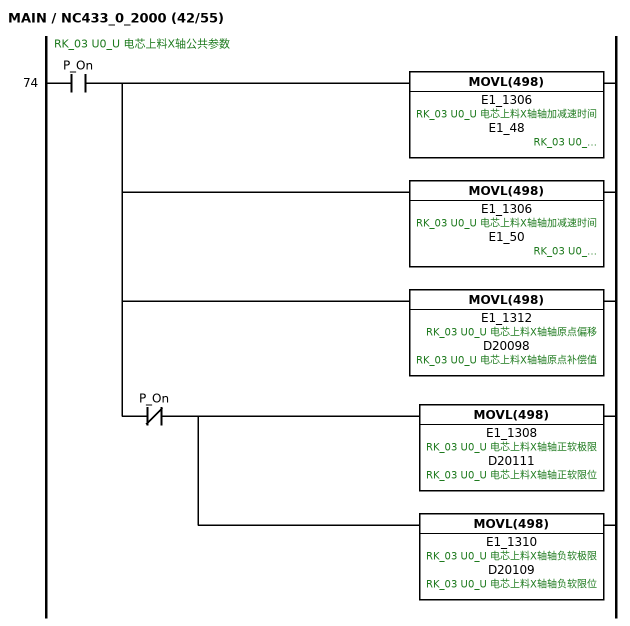
; [picture p96: MAIN / NC433_0_2000, rungs 74-74]
; rung 74: RK_03 U0_U 电芯上料X轴公共参数
LD P_On
MOVL(498) E1_1306 E1_48  ; RK_03 U0_U 电芯上料X轴轴加减速时间, RK_03 U0_U 电芯上料X轴轴直接操作加速时间
MOVL(498) E1_1306 E1_50  ; RK_03 U0_U 电芯上料X轴轴加减速时间, RK_03 U0_U 电芯上料X轴轴直接操作减速时间
MOVL(498) E1_1312 D20098  ; RK_03 U0_U 电芯上料X轴轴原点偏移, RK_03 U0_U 电芯上料X轴轴原点补偿值
ANDNOT P_On
MOVL(498) E1_1308 D20111  ; RK_03 U0_U 电芯上料X轴轴正软极限, RK_03 U0_U 电芯上料X轴轴正软限位
MOVL(498) E1_1310 D20109  ; RK_03 U0_U 电芯上料X轴轴负软极限, RK_03 U0_U 电芯上料X轴轴负软限位

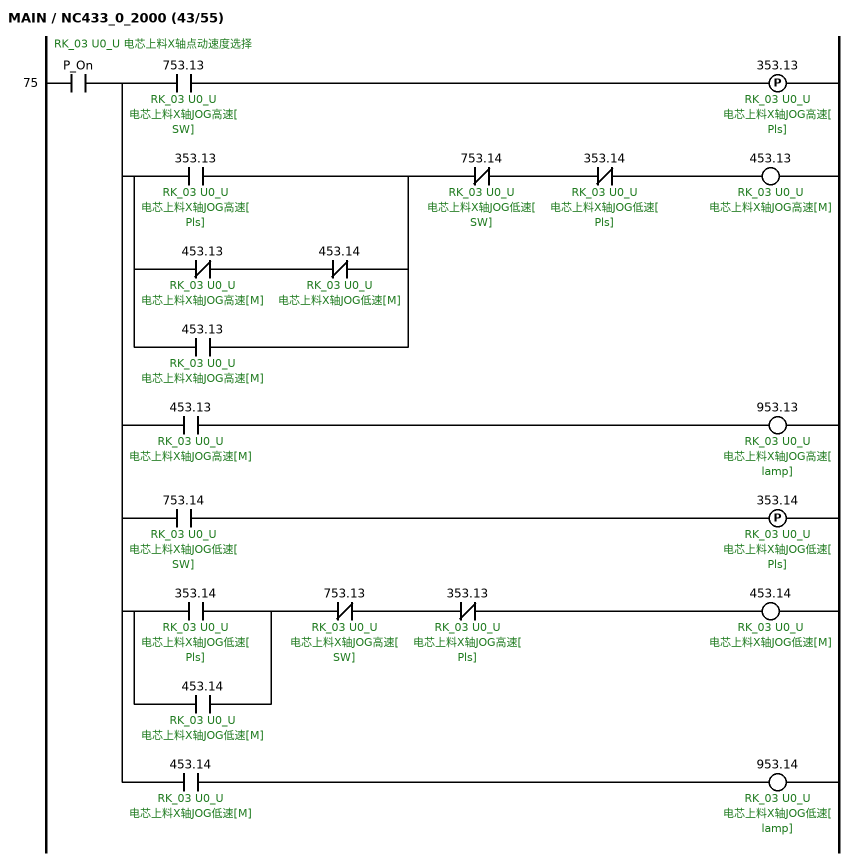
; rung 75: RK_03 U0_U 电芯上料X轴点动速度选择
LD P_On
OUT TR0
AND 753.13  ; RK_03 U0_U 电芯上料X轴JOG高速[SW]
DIFU(013) 353.13  ; RK_03 U0_U 电芯上料X轴JOG高速[Pls]
LD TR0
LD 353.13  ; RK_03 U0_U 电芯上料X轴JOG高速[Pls]
LDNOT 453.13  ; RK_03 U0_U 电芯上料X轴JOG高速[M]
ANDNOT 453.14  ; RK_03 U0_U 电芯上料X轴JOG低速[M]
ORLD
OR 453.13  ; RK_03 U0_U 电芯上料X轴JOG高速[M]
ANDLD
ANDNOT 753.14  ; RK_03 U0_U 电芯上料X轴JOG低速[SW]
ANDNOT 353.14  ; RK_03 U0_U 电芯上料X轴JOG低速[Pls]
OUT 453.13  ; RK_03 U0_U 电芯上料X轴JOG高速[M]
LD TR0
AND 453.13  ; RK_03 U0_U 电芯上料X轴JOG高速[M]
OUT 953.13  ; RK_03 U0_U 电芯上料X轴JOG高速[lamp]
LD TR0
AND 753.14  ; RK_03 U0_U 电芯上料X轴JOG低速[SW]
DIFU(013) 353.14  ; RK_03 U0_U 电芯上料X轴JOG低速[Pls]
LD TR0
LD 353.14  ; RK_03 U0_U 电芯上料X轴JOG低速[Pls]
OR 453.14  ; RK_03 U0_U 电芯上料X轴JOG低速[M]
ANDLD
ANDNOT 753.13  ; RK_03 U0_U 电芯上料X轴JOG高速[SW]
ANDNOT 353.13  ; RK_03 U0_U 电芯上料X轴JOG高速[Pls]
OUT 453.14  ; RK_03 U0_U 电芯上料X轴JOG低速[M]
LD TR0
AND 453.14  ; RK_03 U0_U 电芯上料X轴JOG低速[M]
OUT 953.14  ; RK_03 U0_U 电芯上料X轴JOG低速[lamp]

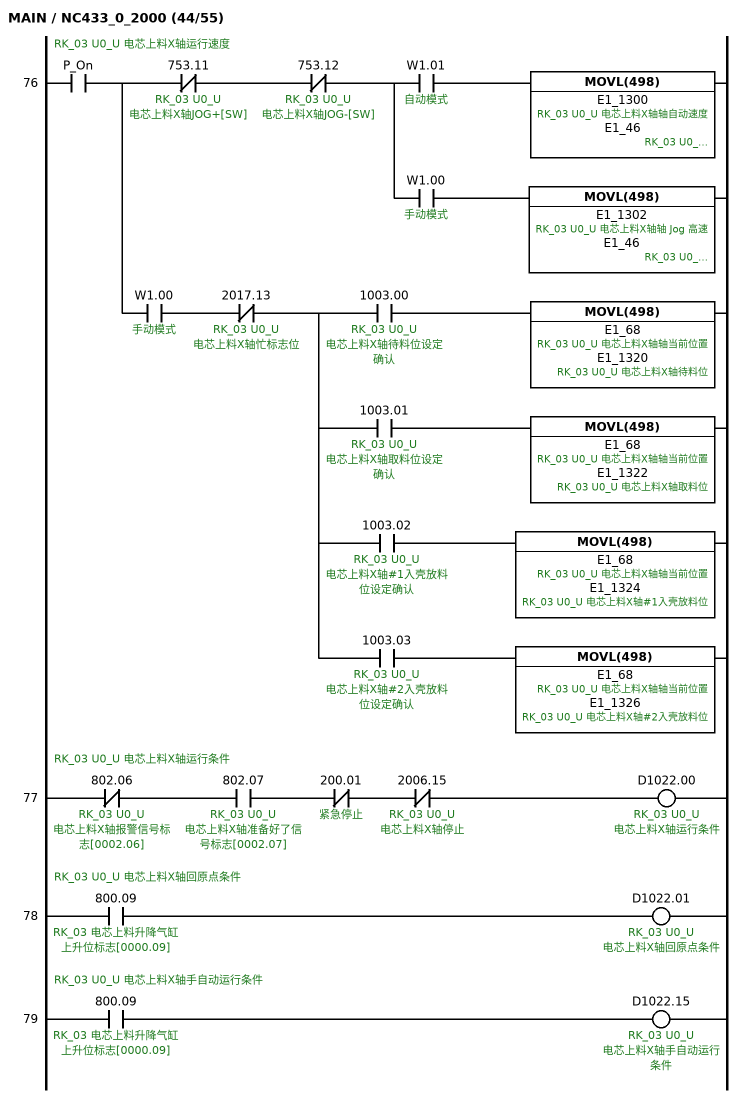
; rung 76: RK_03 U0_U 电芯上料X轴运行速度
LD P_On
OUT TR0
ANDNOT 753.11  ; RK_03 U0_U 电芯上料X轴JOG+[SW]
ANDNOT 753.12  ; RK_03 U0_U 电芯上料X轴JOG-[SW]
OUT TR1
AND W1.01  ; 自动模式
MOVL(498) E1_1300 E1_46  ; RK_03 U0_U 电芯上料X轴轴自动速度, RK_03 U0_U 电芯上料X轴轴直接操作速度
LD TR1
AND W1.00  ; 手动模式
MOVL(498) E1_1302 E1_46  ; RK_03 U0_U 电芯上料X轴轴 Jog 高速, RK_03 U0_U 电芯上料X轴轴直接操作速度
LD TR0
AND W1.00  ; 手动模式
ANDNOT 2017.13  ; RK_03 U0_U 电芯上料X轴忙标志位
OUT TR0
AND 1003.00  ; RK_03 U0_U 电芯上料X轴待料位设定确认
MOVL(498) E1_68 E1_1320  ; RK_03 U0_U 电芯上料X轴轴当前位置, RK_03 U0_U 电芯上料X轴待料位
LD TR0
AND 1003.01  ; RK_03 U0_U 电芯上料X轴取料位设定确认
MOVL(498) E1_68 E1_1322  ; RK_03 U0_U 电芯上料X轴轴当前位置, RK_03 U0_U 电芯上料X轴取料位
LD TR0
AND 1003.02  ; RK_03 U0_U 电芯上料X轴#1入壳放料位设定确认
MOVL(498) E1_68 E1_1324  ; RK_03 U0_U 电芯上料X轴轴当前位置, RK_03 U0_U 电芯上料X轴#1入壳放料位
LD TR0
AND 1003.03  ; RK_03 U0_U 电芯上料X轴#2入壳放料位设定确认
MOVL(498) E1_68 E1_1326  ; RK_03 U0_U 电芯上料X轴轴当前位置, RK_03 U0_U 电芯上料X轴#2入壳放料位
; rung 77: RK_03 U0_U 电芯上料X轴运行条件
LDNOT 802.06  ; RK_03 U0_U 电芯上料X轴报警信号标志[0002.06]
AND 802.07  ; RK_03 U0_U 电芯上料X轴准备好了信号标志[0002.07]
ANDNOT 200.01  ; 紧急停止
ANDNOT 2006.15  ; RK_03 U0_U 电芯上料X轴停止
OUT D1022.00  ; RK_03 U0_U 电芯上料X轴运行条件
; rung 78: RK_03 U0_U 电芯上料X轴回原点条件
LD 800.09  ; RK_03 电芯上料升降气缸上升位标志[0000.09]
OUT D1022.01  ; RK_03 U0_U 电芯上料X轴回原点条件
; rung 79: RK_03 U0_U 电芯上料X轴手自动运行条件
LD 800.09  ; RK_03 电芯上料升降气缸上升位标志[0000.09]
OUT D1022.15  ; RK_03 U0_U 电芯上料X轴手自动运行条件

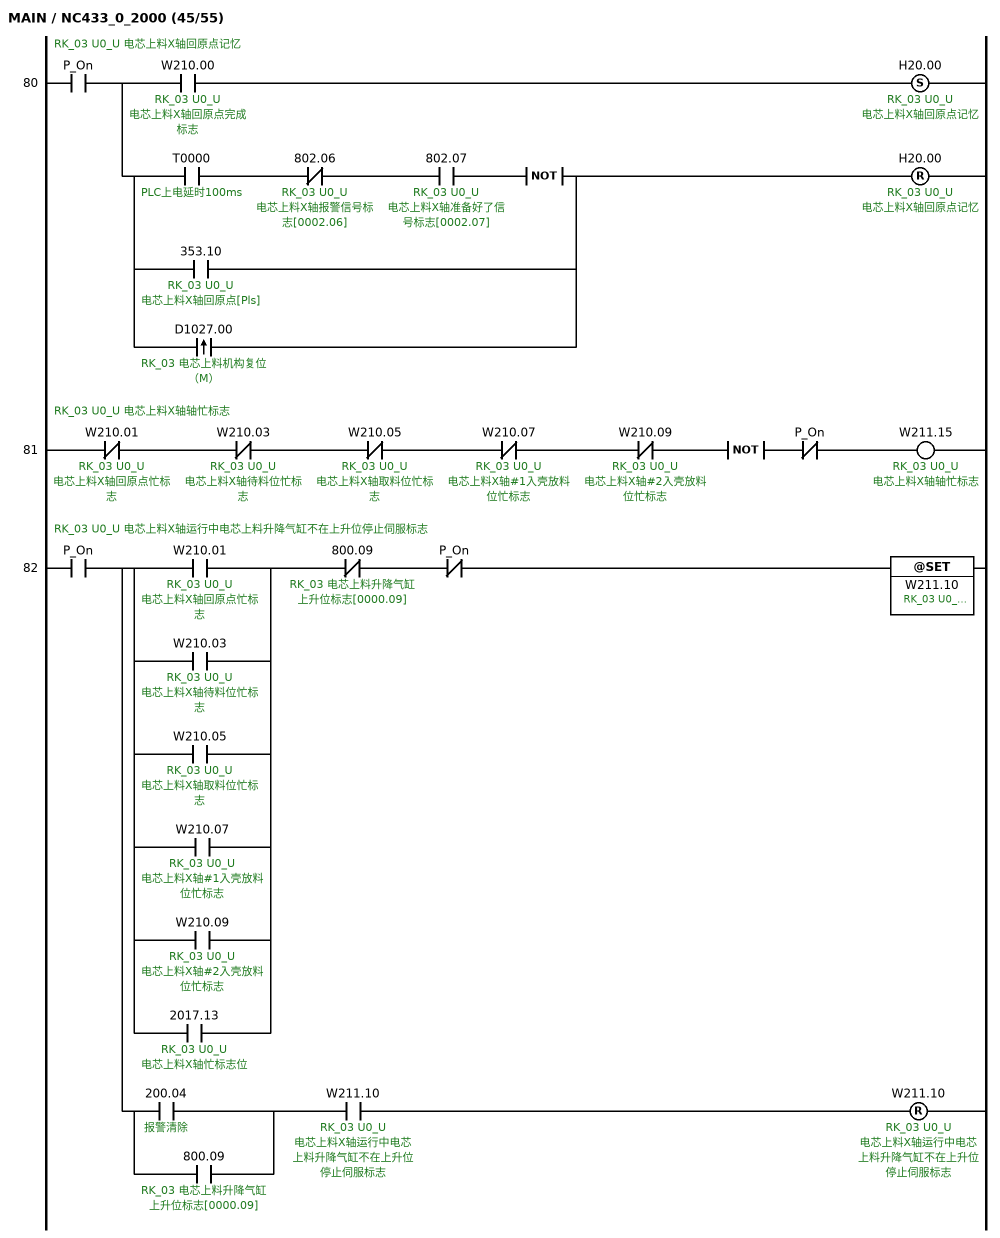
; rung 80: RK_03 U0_U 电芯上料X轴回原点记忆
LD P_On
OUT TR0
AND W210.00  ; RK_03 U0_U 电芯上料X轴回原点完成标志
SET H20.00  ; RK_03 U0_U 电芯上料X轴回原点记忆
LD TR0
LD T0000  ; PLC上电延时100ms
ANDNOT 802.06  ; RK_03 U0_U 电芯上料X轴报警信号标志[0002.06]
AND 802.07  ; RK_03 U0_U 电芯上料X轴准备好了信号标志[0002.07]
NOT(520)
OR 353.10  ; RK_03 U0_U 电芯上料X轴回原点[Pls]
@OR D1027.00  ; RK_03 电芯上料机构复位（M）
ANDLD
RSET H20.00  ; RK_03 U0_U 电芯上料X轴回原点记忆
; rung 81: RK_03 U0_U 电芯上料X轴轴忙标志
LDNOT W210.01  ; RK_03 U0_U 电芯上料X轴回原点忙标志
ANDNOT W210.03  ; RK_03 U0_U 电芯上料X轴待料位忙标志
ANDNOT W210.05  ; RK_03 U0_U 电芯上料X轴取料位忙标志
ANDNOT W210.07  ; RK_03 U0_U 电芯上料X轴#1入壳放料位忙标志
ANDNOT W210.09  ; RK_03 U0_U 电芯上料X轴#2入壳放料位忙标志
NOT(520)
ANDNOT P_On
OUT W211.15  ; RK_03 U0_U 电芯上料X轴轴忙标志
; rung 82: RK_03 U0_U 电芯上料X轴运行中电芯上料升降气缸不在上升位停止伺服标志
LD P_On
OUT TR0
LD W210.01  ; RK_03 U0_U 电芯上料X轴回原点忙标志
OR W210.03  ; RK_03 U0_U 电芯上料X轴待料位忙标志
OR W210.05  ; RK_03 U0_U 电芯上料X轴取料位忙标志
OR W210.07  ; RK_03 U0_U 电芯上料X轴#1入壳放料位忙标志
OR W210.09  ; RK_03 U0_U 电芯上料X轴#2入壳放料位忙标志
OR 2017.13  ; RK_03 U0_U 电芯上料X轴忙标志位
ANDLD
ANDNOT 800.09  ; RK_03 电芯上料升降气缸上升位标志[0000.09]
ANDNOT P_On
@SET W211.10  ; RK_03 U0_U 电芯上料X轴运行中电芯上料升降气缸不在上升位停止伺服标志  // 增加相应报警信息
LD TR0
LD 200.04  ; 报警清除
OR 800.09  ; RK_03 电芯上料升降气缸上升位标志[0000.09]
ANDLD
AND W211.10  ; RK_03 U0_U 电芯上料X轴运行中电芯上料升降气缸不在上升位停止伺服标志
RSET W211.10  ; RK_03 U0_U 电芯上料X轴运行中电芯上料升降气缸不在上升位停止伺服标志

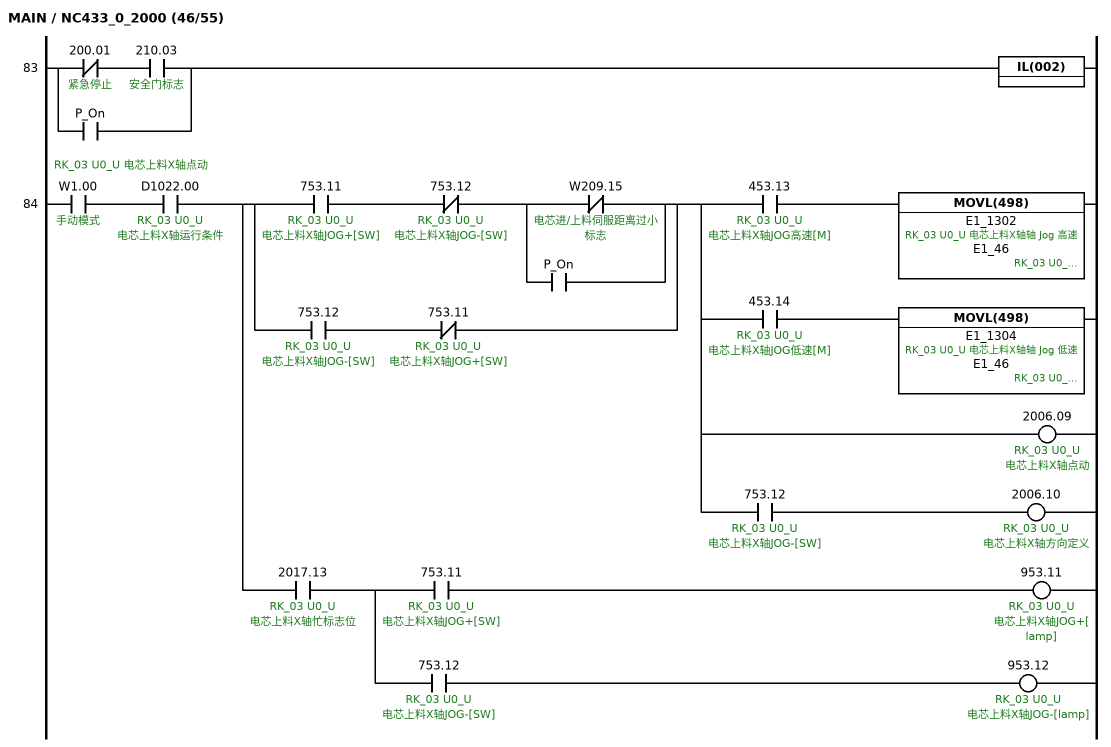
; rung 83
LDNOT 200.01  ; 紧急停止
AND 210.03  ; 安全门标志
OR P_On
IL(002)
; rung 84: RK_03 U0_U 电芯上料X轴点动
LD W1.00  ; 手动模式
AND D1022.00  ; RK_03 U0_U 电芯上料X轴运行条件
OUT TR0
LD 753.11  ; RK_03 U0_U 电芯上料X轴JOG+[SW]
ANDNOT 753.12  ; RK_03 U0_U 电芯上料X轴JOG-[SW]
LDNOT W209.15  ; 电芯进/上料伺服距离过小标志
OR P_On
ANDLD
LD 753.12  ; RK_03 U0_U 电芯上料X轴JOG-[SW]
ANDNOT 753.11  ; RK_03 U0_U 电芯上料X轴JOG+[SW]
ORLD
ANDLD
OUT TR1
AND 453.13  ; RK_03 U0_U 电芯上料X轴JOG高速[M]
MOVL(498) E1_1302 E1_46  ; RK_03 U0_U 电芯上料X轴轴 Jog 高速, RK_03 U0_U 电芯上料X轴轴直接操作速度
LD TR1
AND 453.14  ; RK_03 U0_U 电芯上料X轴JOG低速[M]
MOVL(498) E1_1304 E1_46  ; RK_03 U0_U 电芯上料X轴轴 Jog 低速, RK_03 U0_U 电芯上料X轴轴直接操作速度
LD TR1
OUT 2006.09  ; RK_03 U0_U 电芯上料X轴点动
AND 753.12  ; RK_03 U0_U 电芯上料X轴JOG-[SW]
OUT 2006.10  ; RK_03 U0_U 电芯上料X轴方向定义
LD TR0
AND 2017.13  ; RK_03 U0_U 电芯上料X轴忙标志位
OUT TR0
AND 753.11  ; RK_03 U0_U 电芯上料X轴JOG+[SW]
OUT 953.11  ; RK_03 U0_U 电芯上料X轴JOG+[lamp]
LD TR0
AND 753.12  ; RK_03 U0_U 电芯上料X轴JOG-[SW]
OUT 953.12  ; RK_03 U0_U 电芯上料X轴JOG-[lamp]

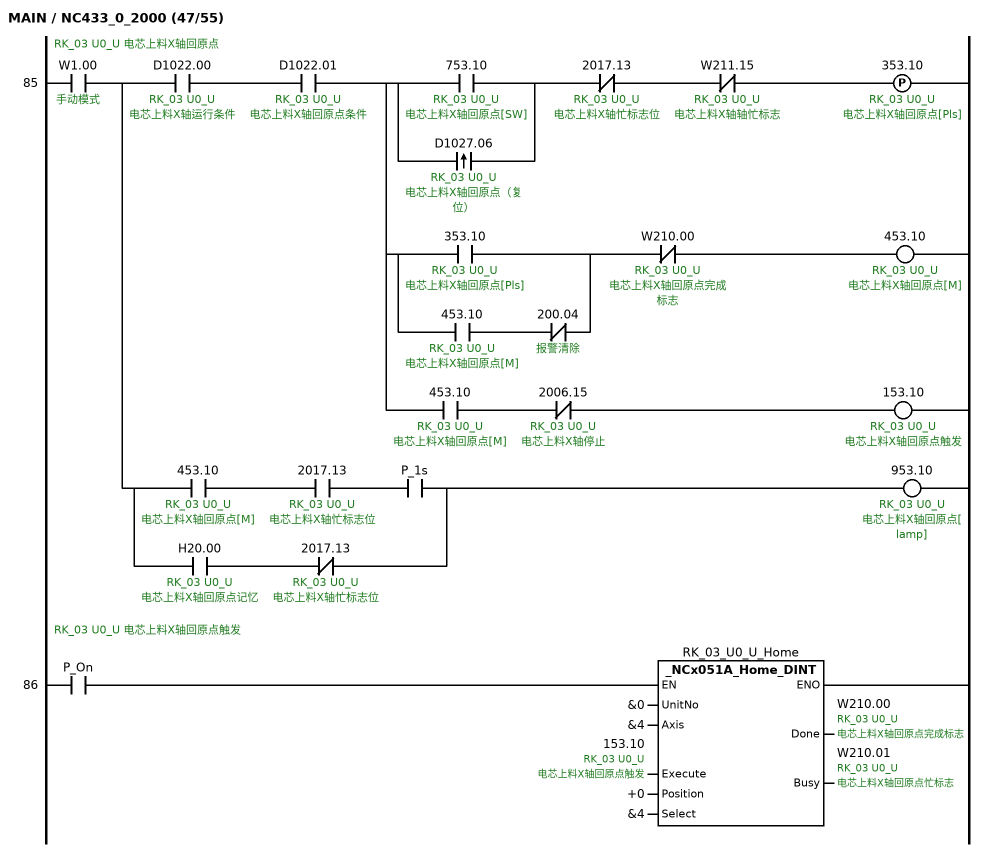
; rung 85: RK_03 U0_U 电芯上料X轴回原点
LD W1.00  ; 手动模式
OUT TR0
AND D1022.00  ; RK_03 U0_U 电芯上料X轴运行条件
AND D1022.01  ; RK_03 U0_U 电芯上料X轴回原点条件
OUT TR1
LD 753.10  ; RK_03 U0_U 电芯上料X轴回原点[SW]
@OR D1027.06  ; RK_03 U0_U 电芯上料X轴回原点（复位）
ANDLD
ANDNOT 2017.13  ; RK_03 U0_U 电芯上料X轴忙标志位
ANDNOT W211.15  ; RK_03 U0_U 电芯上料X轴轴忙标志
DIFU(013) 353.10  ; RK_03 U0_U 电芯上料X轴回原点[Pls]
LD TR1
LD 353.10  ; RK_03 U0_U 电芯上料X轴回原点[Pls]
LD 453.10  ; RK_03 U0_U 电芯上料X轴回原点[M]
ANDNOT 200.04  ; 报警清除
ORLD
ANDLD
ANDNOT W210.00  ; RK_03 U0_U 电芯上料X轴回原点完成标志
OUT 453.10  ; RK_03 U0_U 电芯上料X轴回原点[M]
LD TR1
AND 453.10  ; RK_03 U0_U 电芯上料X轴回原点[M]
ANDNOT 2006.15  ; RK_03 U0_U 电芯上料X轴停止
OUT 153.10  ; RK_03 U0_U 电芯上料X轴回原点触发
LD TR0
LD 453.10  ; RK_03 U0_U 电芯上料X轴回原点[M]
AND 2017.13  ; RK_03 U0_U 电芯上料X轴忙标志位
AND P_1s
LD H20.00  ; RK_03 U0_U 电芯上料X轴回原点记忆
ANDNOT 2017.13  ; RK_03 U0_U 电芯上料X轴忙标志位
ORLD
ANDLD
OUT 953.10  ; RK_03 U0_U 电芯上料X轴回原点[lamp]
; rung 86: RK_03 U0_U 电芯上料X轴回原点触发
LD P_On
CALL RK_03_U0_U_Home : _NCx051A_Home_DINT (UnitNo := &0, Axis := &4, Execute := 153.10, Position := +0, Select := &4, Done => W210.00, Busy => W210.01)  ; RK_03 U0_U 电芯上料X轴回原点触发, RK_03 U0_U 电芯上料X轴回原点完成标志, RK_03 U0_U 电芯上料X轴回原点忙标志

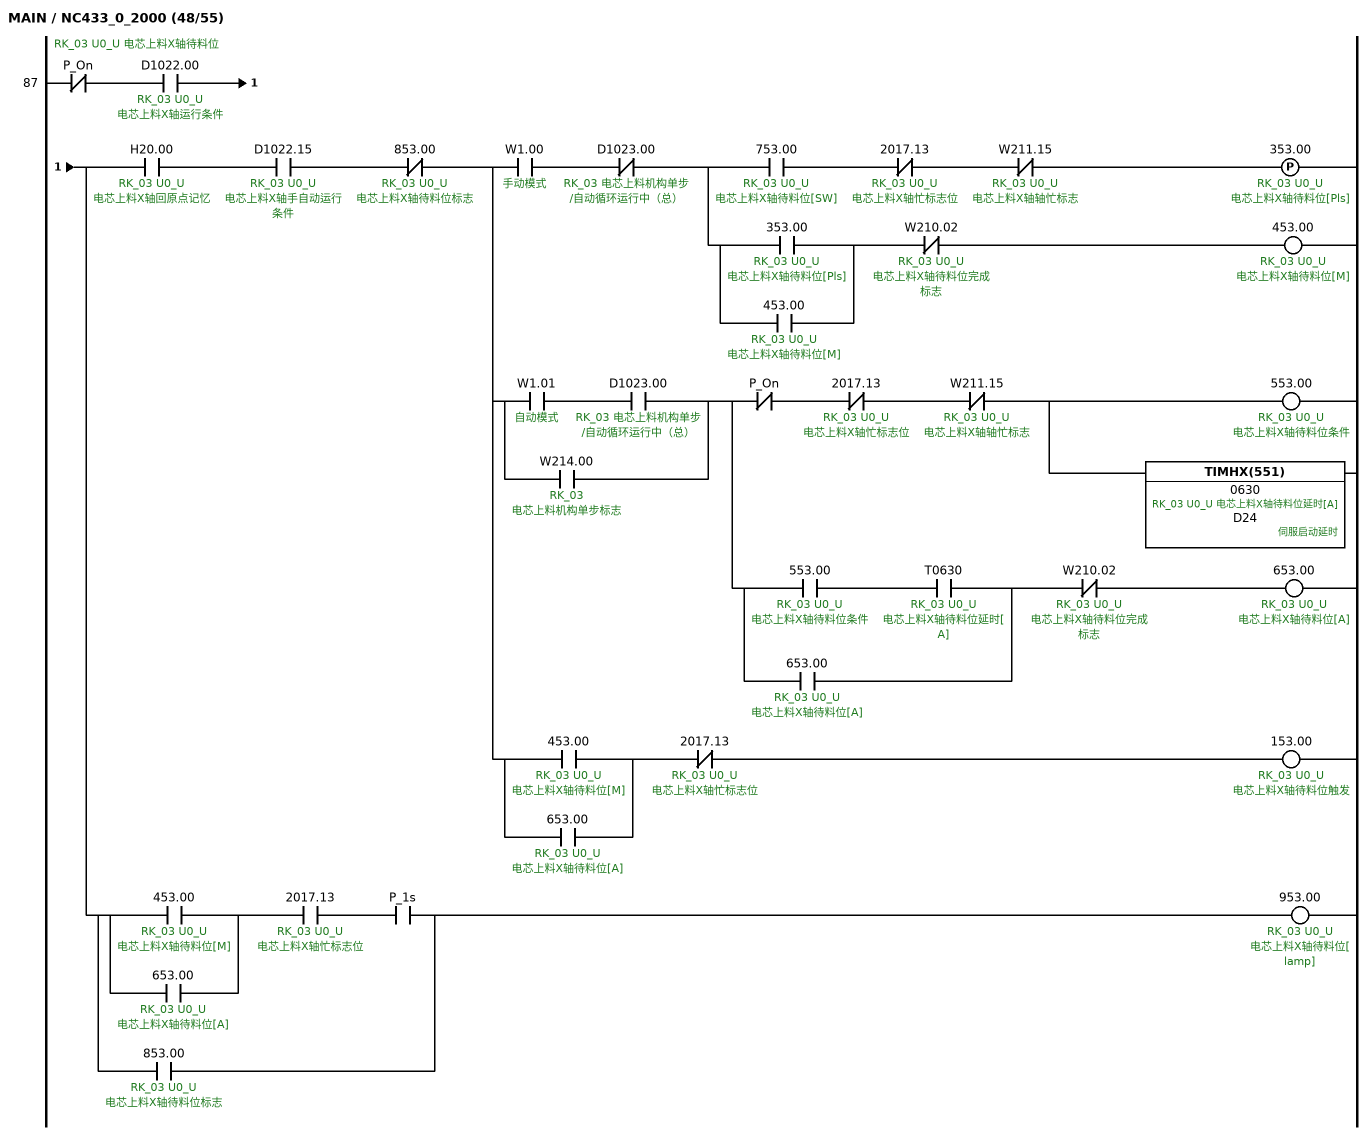
; rung 87: RK_03 U0_U 电芯上料X轴待料位
LDNOT P_On
AND D1022.00  ; RK_03 U0_U 电芯上料X轴运行条件
OUT TR0
AND H20.00  ; RK_03 U0_U 电芯上料X轴回原点记忆
AND D1022.15  ; RK_03 U0_U 电芯上料X轴手自动运行条件
ANDNOT 853.00  ; RK_03 U0_U 电芯上料X轴待料位标志
OUT TR1
AND W1.00  ; 手动模式
ANDNOT D1023.00  ; RK_03 电芯上料机构单步/自动循环运行中（总）
OUT TR2
AND 753.00  ; RK_03 U0_U 电芯上料X轴待料位[SW]
ANDNOT 2017.13  ; RK_03 U0_U 电芯上料X轴忙标志位
ANDNOT W211.15  ; RK_03 U0_U 电芯上料X轴轴忙标志
DIFU(013) 353.00  ; RK_03 U0_U 电芯上料X轴待料位[Pls]
LD TR2
LD 353.00  ; RK_03 U0_U 电芯上料X轴待料位[Pls]
OR 453.00  ; RK_03 U0_U 电芯上料X轴待料位[M]
ANDLD
ANDNOT W210.02  ; RK_03 U0_U 电芯上料X轴待料位完成标志
OUT 453.00  ; RK_03 U0_U 电芯上料X轴待料位[M]
LD TR1
LD W1.01  ; 自动模式
AND D1023.00  ; RK_03 电芯上料机构单步/自动循环运行中（总）
OR W214.00  ; RK_03  电芯上料机构单步标志
ANDLD
OUT TR2
ANDNOT P_On  // RK_03 U0_U 电芯上料X轴待料位
ANDNOT 2017.13  ; RK_03 U0_U 电芯上料X轴忙标志位
ANDNOT W211.15  ; RK_03 U0_U 电芯上料X轴轴忙标志
OUT 553.00  ; RK_03 U0_U 电芯上料X轴待料位条件
TIMHX(551) 0630 D24  ; 伺服启动延时, RK_03 U0_U 电芯上料X轴待料位延时[A]
LD TR2
LD 553.00  ; RK_03 U0_U 电芯上料X轴待料位条件
AND T0630  ; RK_03 U0_U 电芯上料X轴待料位延时[A]
OR 653.00  ; RK_03 U0_U 电芯上料X轴待料位[A]
ANDLD
ANDNOT W210.02  ; RK_03 U0_U 电芯上料X轴待料位完成标志
OUT 653.00  ; RK_03 U0_U 电芯上料X轴待料位[A]
LD TR1
LD 453.00  ; RK_03 U0_U 电芯上料X轴待料位[M]
OR 653.00  ; RK_03 U0_U 电芯上料X轴待料位[A]
ANDLD
ANDNOT 2017.13  ; RK_03 U0_U 电芯上料X轴忙标志位
OUT 153.00  ; RK_03 U0_U 电芯上料X轴待料位触发
LD TR0
LD 453.00  ; RK_03 U0_U 电芯上料X轴待料位[M]
OR 653.00  ; RK_03 U0_U 电芯上料X轴待料位[A]
AND 2017.13  ; RK_03 U0_U 电芯上料X轴忙标志位
AND P_1s
OR 853.00  ; RK_03 U0_U 电芯上料X轴待料位标志
ANDLD
OUT 953.00  ; RK_03 U0_U 电芯上料X轴待料位[lamp]

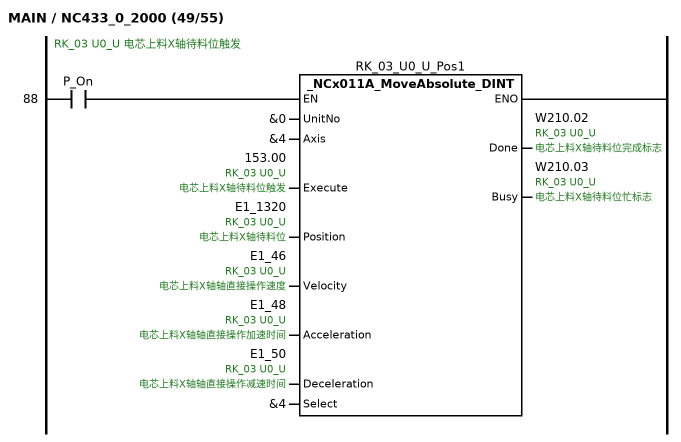
; rung 88: RK_03 U0_U 电芯上料X轴待料位触发
LD P_On
CALL RK_03_U0_U_Pos1 : _NCx011A_MoveAbsolute_DINT (UnitNo := &0, Axis := &4, Execute := 153.00, Position := E1_1320, Velocity := E1_46, Acceleration := E1_48, Deceleration := E1_50, Select := &4, Done => W210.02, Busy => W210.03)  ; RK_03 U0_U 电芯上料X轴待料位触发, RK_03 U0_U 电芯上料X轴待料位, RK_03 U0_U 电芯上料X轴轴直接操作速度, RK_03 U0_U 电芯上料X轴轴直接操作加速时间, RK_03 U0_U 电芯上料X轴轴直接操作减速时间, RK_03 U0_U 电芯上料X轴待料位完成标志, RK_03 U0_U 电芯上料X轴待料位忙标志

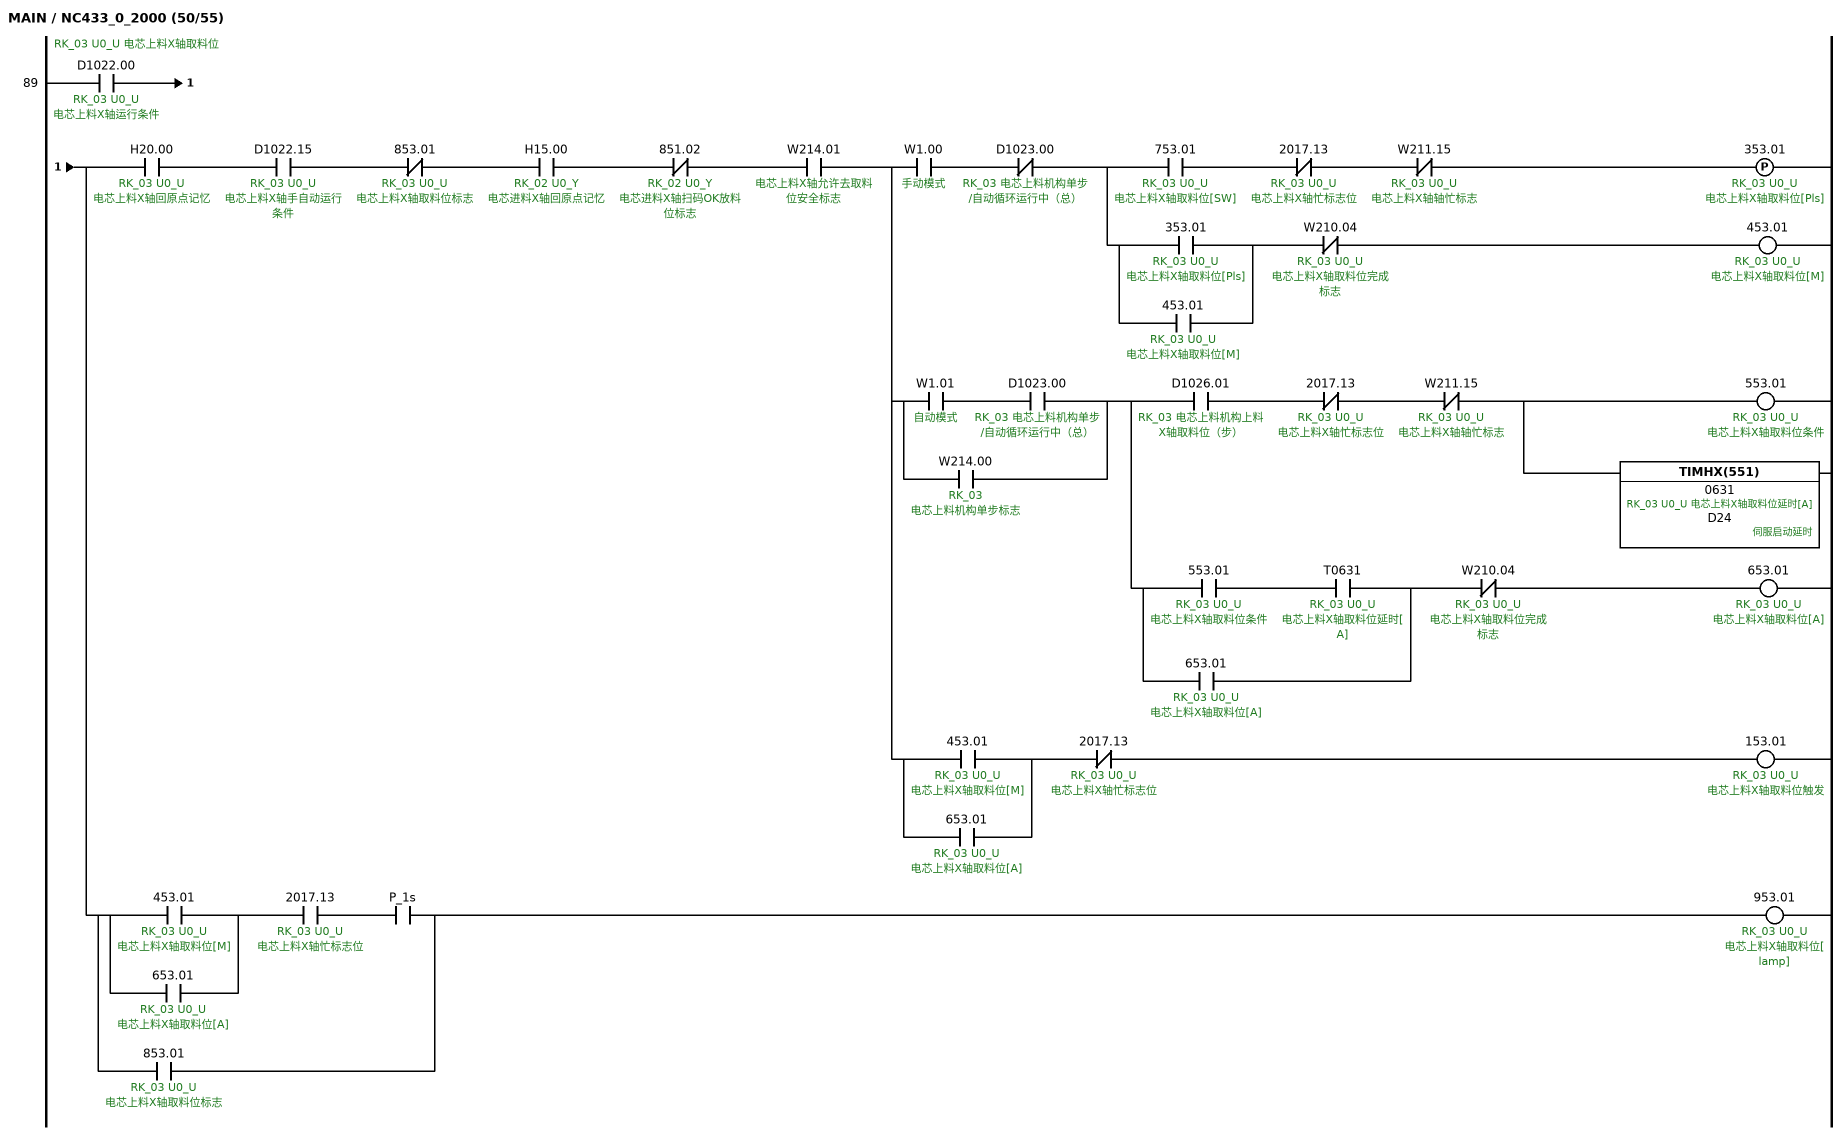
; rung 89: RK_03 U0_U 电芯上料X轴取料位
LD D1022.00  ; RK_03 U0_U 电芯上料X轴运行条件
OUT TR0
AND H20.00  ; RK_03 U0_U 电芯上料X轴回原点记忆
AND D1022.15  ; RK_03 U0_U 电芯上料X轴手自动运行条件
ANDNOT 853.01  ; RK_03 U0_U 电芯上料X轴取料位标志
AND H15.00  ; RK_02 U0_Y 电芯进料X轴回原点记忆
ANDNOT 851.02  ; RK_02 U0_Y 电芯进料X轴扫码OK放料位标志
AND W214.01  ; 电芯上料X轴允许去取料位安全标志
OUT TR1
AND W1.00  ; 手动模式
ANDNOT D1023.00  ; RK_03 电芯上料机构单步/自动循环运行中（总）
OUT TR2
AND 753.01  ; RK_03 U0_U 电芯上料X轴取料位[SW]
ANDNOT 2017.13  ; RK_03 U0_U 电芯上料X轴忙标志位
ANDNOT W211.15  ; RK_03 U0_U 电芯上料X轴轴忙标志
DIFU(013) 353.01  ; RK_03 U0_U 电芯上料X轴取料位[Pls]
LD TR2
LD 353.01  ; RK_03 U0_U 电芯上料X轴取料位[Pls]
OR 453.01  ; RK_03 U0_U 电芯上料X轴取料位[M]
ANDLD
ANDNOT W210.04  ; RK_03 U0_U 电芯上料X轴取料位完成标志
OUT 453.01  ; RK_03 U0_U 电芯上料X轴取料位[M]
LD TR1
LD W1.01  ; 自动模式
AND D1023.00  ; RK_03 电芯上料机构单步/自动循环运行中（总）
OR W214.00  ; RK_03  电芯上料机构单步标志
ANDLD
OUT TR2
AND D1026.01  ; RK_03 电芯上料机构上料X轴取料位（步）
ANDNOT 2017.13  ; RK_03 U0_U 电芯上料X轴忙标志位
ANDNOT W211.15  ; RK_03 U0_U 电芯上料X轴轴忙标志
OUT 553.01  ; RK_03 U0_U 电芯上料X轴取料位条件
TIMHX(551) 0631 D24  ; 伺服启动延时, RK_03 U0_U 电芯上料X轴取料位延时[A]
LD TR2
LD 553.01  ; RK_03 U0_U 电芯上料X轴取料位条件
AND T0631  ; RK_03 U0_U 电芯上料X轴取料位延时[A]
OR 653.01  ; RK_03 U0_U 电芯上料X轴取料位[A]
ANDLD
ANDNOT W210.04  ; RK_03 U0_U 电芯上料X轴取料位完成标志
OUT 653.01  ; RK_03 U0_U 电芯上料X轴取料位[A]
LD TR1
LD 453.01  ; RK_03 U0_U 电芯上料X轴取料位[M]
OR 653.01  ; RK_03 U0_U 电芯上料X轴取料位[A]
ANDLD
ANDNOT 2017.13  ; RK_03 U0_U 电芯上料X轴忙标志位
OUT 153.01  ; RK_03 U0_U 电芯上料X轴取料位触发
LD TR0
LD 453.01  ; RK_03 U0_U 电芯上料X轴取料位[M]
OR 653.01  ; RK_03 U0_U 电芯上料X轴取料位[A]
AND 2017.13  ; RK_03 U0_U 电芯上料X轴忙标志位
AND P_1s
OR 853.01  ; RK_03 U0_U 电芯上料X轴取料位标志
ANDLD
OUT 953.01  ; RK_03 U0_U 电芯上料X轴取料位[lamp]

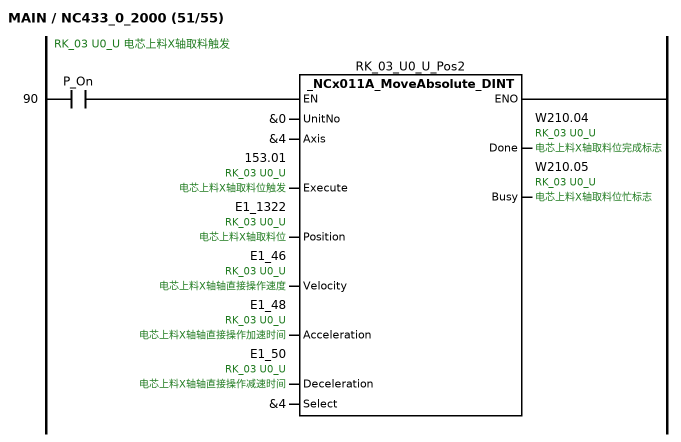
; rung 90: RK_03 U0_U 电芯上料X轴取料触发
LD P_On
CALL RK_03_U0_U_Pos2 : _NCx011A_MoveAbsolute_DINT (UnitNo := &0, Axis := &4, Execute := 153.01, Position := E1_1322, Velocity := E1_46, Acceleration := E1_48, Deceleration := E1_50, Select := &4, Done => W210.04, Busy => W210.05)  ; RK_03 U0_U 电芯上料X轴取料位触发, RK_03 U0_U 电芯上料X轴取料位, RK_03 U0_U 电芯上料X轴轴直接操作速度, RK_03 U0_U 电芯上料X轴轴直接操作加速时间, RK_03 U0_U 电芯上料X轴轴直接操作减速时间, RK_03 U0_U 电芯上料X轴取料位完成标志, RK_03 U0_U 电芯上料X轴取料位忙标志

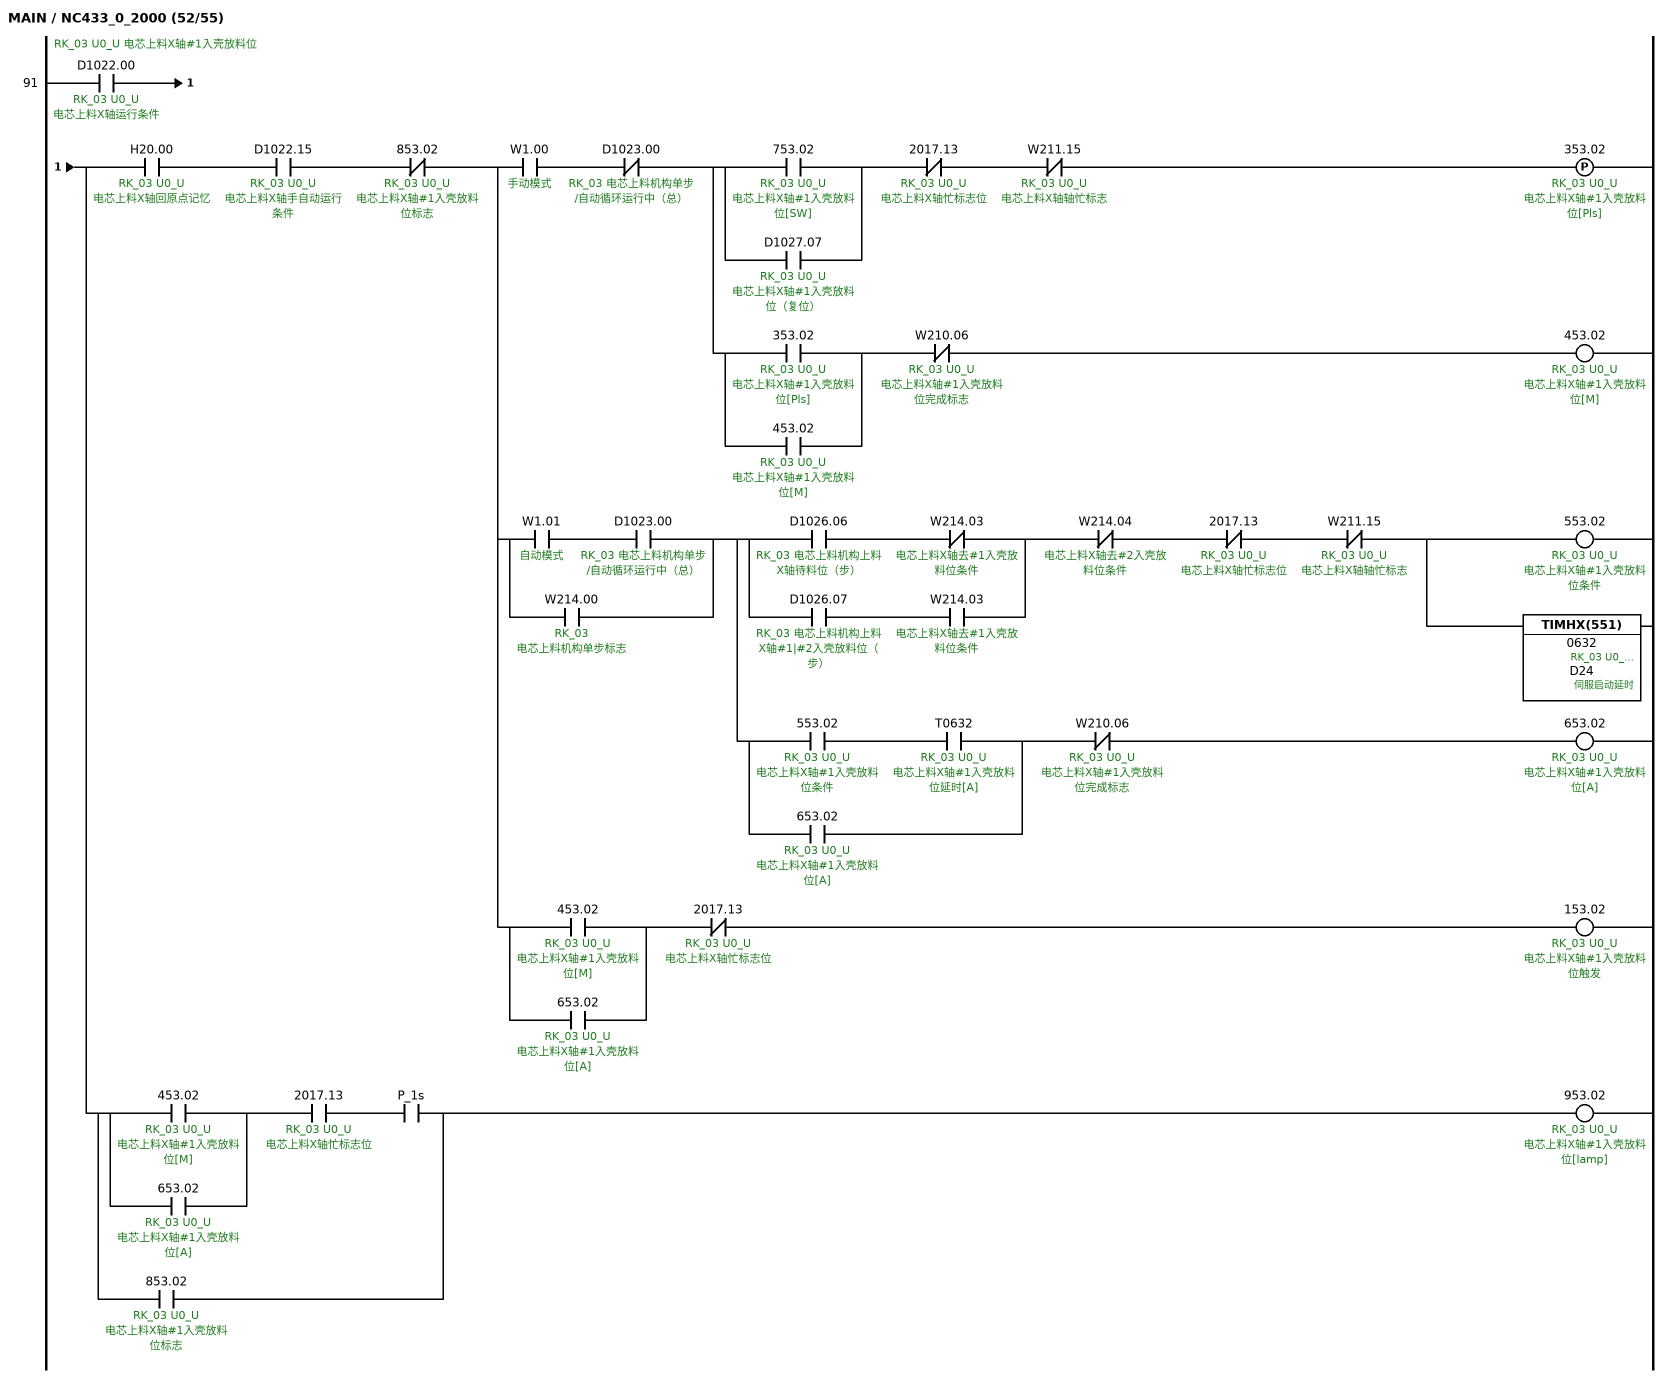
; rung 91: RK_03 U0_U 电芯上料X轴#1入壳放料位
LD D1022.00  ; RK_03 U0_U 电芯上料X轴运行条件
OUT TR0
AND H20.00  ; RK_03 U0_U 电芯上料X轴回原点记忆
AND D1022.15  ; RK_03 U0_U 电芯上料X轴手自动运行条件
ANDNOT 853.02  ; RK_03 U0_U 电芯上料X轴#1入壳放料位标志
OUT TR1
AND W1.00  ; 手动模式
ANDNOT D1023.00  ; RK_03 电芯上料机构单步/自动循环运行中（总）
OUT TR2
LD 753.02  ; RK_03 U0_U 电芯上料X轴#1入壳放料位[SW]
OR D1027.07  ; RK_03 U0_U 电芯上料X轴#1入壳放料位（复位）
ANDLD
ANDNOT 2017.13  ; RK_03 U0_U 电芯上料X轴忙标志位
ANDNOT W211.15  ; RK_03 U0_U 电芯上料X轴轴忙标志
DIFU(013) 353.02  ; RK_03 U0_U 电芯上料X轴#1入壳放料位[Pls]
LD TR2
LD 353.02  ; RK_03 U0_U 电芯上料X轴#1入壳放料位[Pls]
OR 453.02  ; RK_03 U0_U 电芯上料X轴#1入壳放料位[M]
ANDLD
ANDNOT W210.06  ; RK_03 U0_U 电芯上料X轴#1入壳放料位完成标志
OUT 453.02  ; RK_03 U0_U 电芯上料X轴#1入壳放料位[M]
LD TR1
LD W1.01  ; 自动模式
AND D1023.00  ; RK_03 电芯上料机构单步/自动循环运行中（总）
OR W214.00  ; RK_03  电芯上料机构单步标志
ANDLD
OUT TR2
LD D1026.06  ; RK_03 电芯上料机构上料X轴待料位（步）
ANDNOT W214.03  ; 电芯上料X轴去#1入壳放料位条件
LD D1026.07  ; RK_03 电芯上料机构上料X轴#1|#2入壳放料位（步）
AND W214.03  ; 电芯上料X轴去#1入壳放料位条件
ORLD
ANDLD
ANDNOT W214.04  ; 电芯上料X轴去#2入壳放料位条件
ANDNOT 2017.13  ; RK_03 U0_U 电芯上料X轴忙标志位
ANDNOT W211.15  ; RK_03 U0_U 电芯上料X轴轴忙标志
OUT 553.02  ; RK_03 U0_U 电芯上料X轴#1入壳放料位条件
TIMHX(551) 0632 D24  ; 伺服启动延时, RK_03 U0_U 电芯上料X轴#1入壳放料位延时[A]
LD TR2
LD 553.02  ; RK_03 U0_U 电芯上料X轴#1入壳放料位条件
AND T0632  ; RK_03 U0_U 电芯上料X轴#1入壳放料位延时[A]
OR 653.02  ; RK_03 U0_U 电芯上料X轴#1入壳放料位[A]
ANDLD
ANDNOT W210.06  ; RK_03 U0_U 电芯上料X轴#1入壳放料位完成标志
OUT 653.02  ; RK_03 U0_U 电芯上料X轴#1入壳放料位[A]
LD TR1
LD 453.02  ; RK_03 U0_U 电芯上料X轴#1入壳放料位[M]
OR 653.02  ; RK_03 U0_U 电芯上料X轴#1入壳放料位[A]
ANDLD
ANDNOT 2017.13  ; RK_03 U0_U 电芯上料X轴忙标志位
OUT 153.02  ; RK_03 U0_U 电芯上料X轴#1入壳放料位触发
LD TR0
LD 453.02  ; RK_03 U0_U 电芯上料X轴#1入壳放料位[M]
OR 653.02  ; RK_03 U0_U 电芯上料X轴#1入壳放料位[A]
AND 2017.13  ; RK_03 U0_U 电芯上料X轴忙标志位
AND P_1s
OR 853.02  ; RK_03 U0_U 电芯上料X轴#1入壳放料位标志
ANDLD
OUT 953.02  ; RK_03 U0_U 电芯上料X轴#1入壳放料位[lamp]

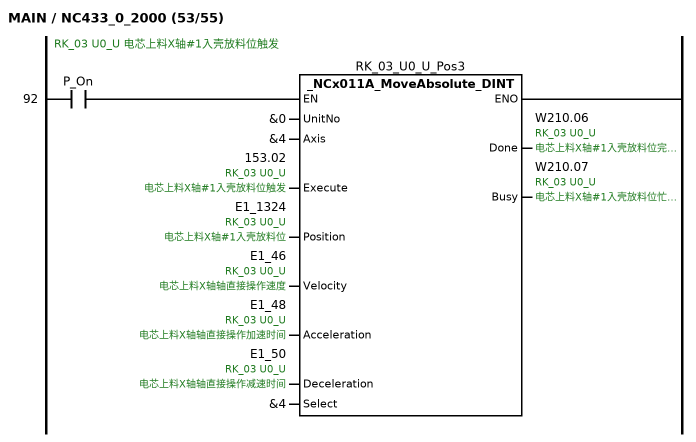
; rung 92: RK_03 U0_U 电芯上料X轴#1入壳放料位触发
LD P_On
CALL RK_03_U0_U_Pos3 : _NCx011A_MoveAbsolute_DINT (UnitNo := &0, Axis := &4, Execute := 153.02, Position := E1_1324, Velocity := E1_46, Acceleration := E1_48, Deceleration := E1_50, Select := &4, Done => W210.06, Busy => W210.07)  ; RK_03 U0_U 电芯上料X轴#1入壳放料位触发, RK_03 U0_U 电芯上料X轴#1入壳放料位, RK_03 U0_U 电芯上料X轴轴直接操作速度, RK_03 U0_U 电芯上料X轴轴直接操作加速时间, RK_03 U0_U 电芯上料X轴轴直接操作减速时间, RK_03 U0_U 电芯上料X轴#1入壳放料位完成标志, RK_03 U0_U 电芯上料X轴#1入壳放料位忙标志

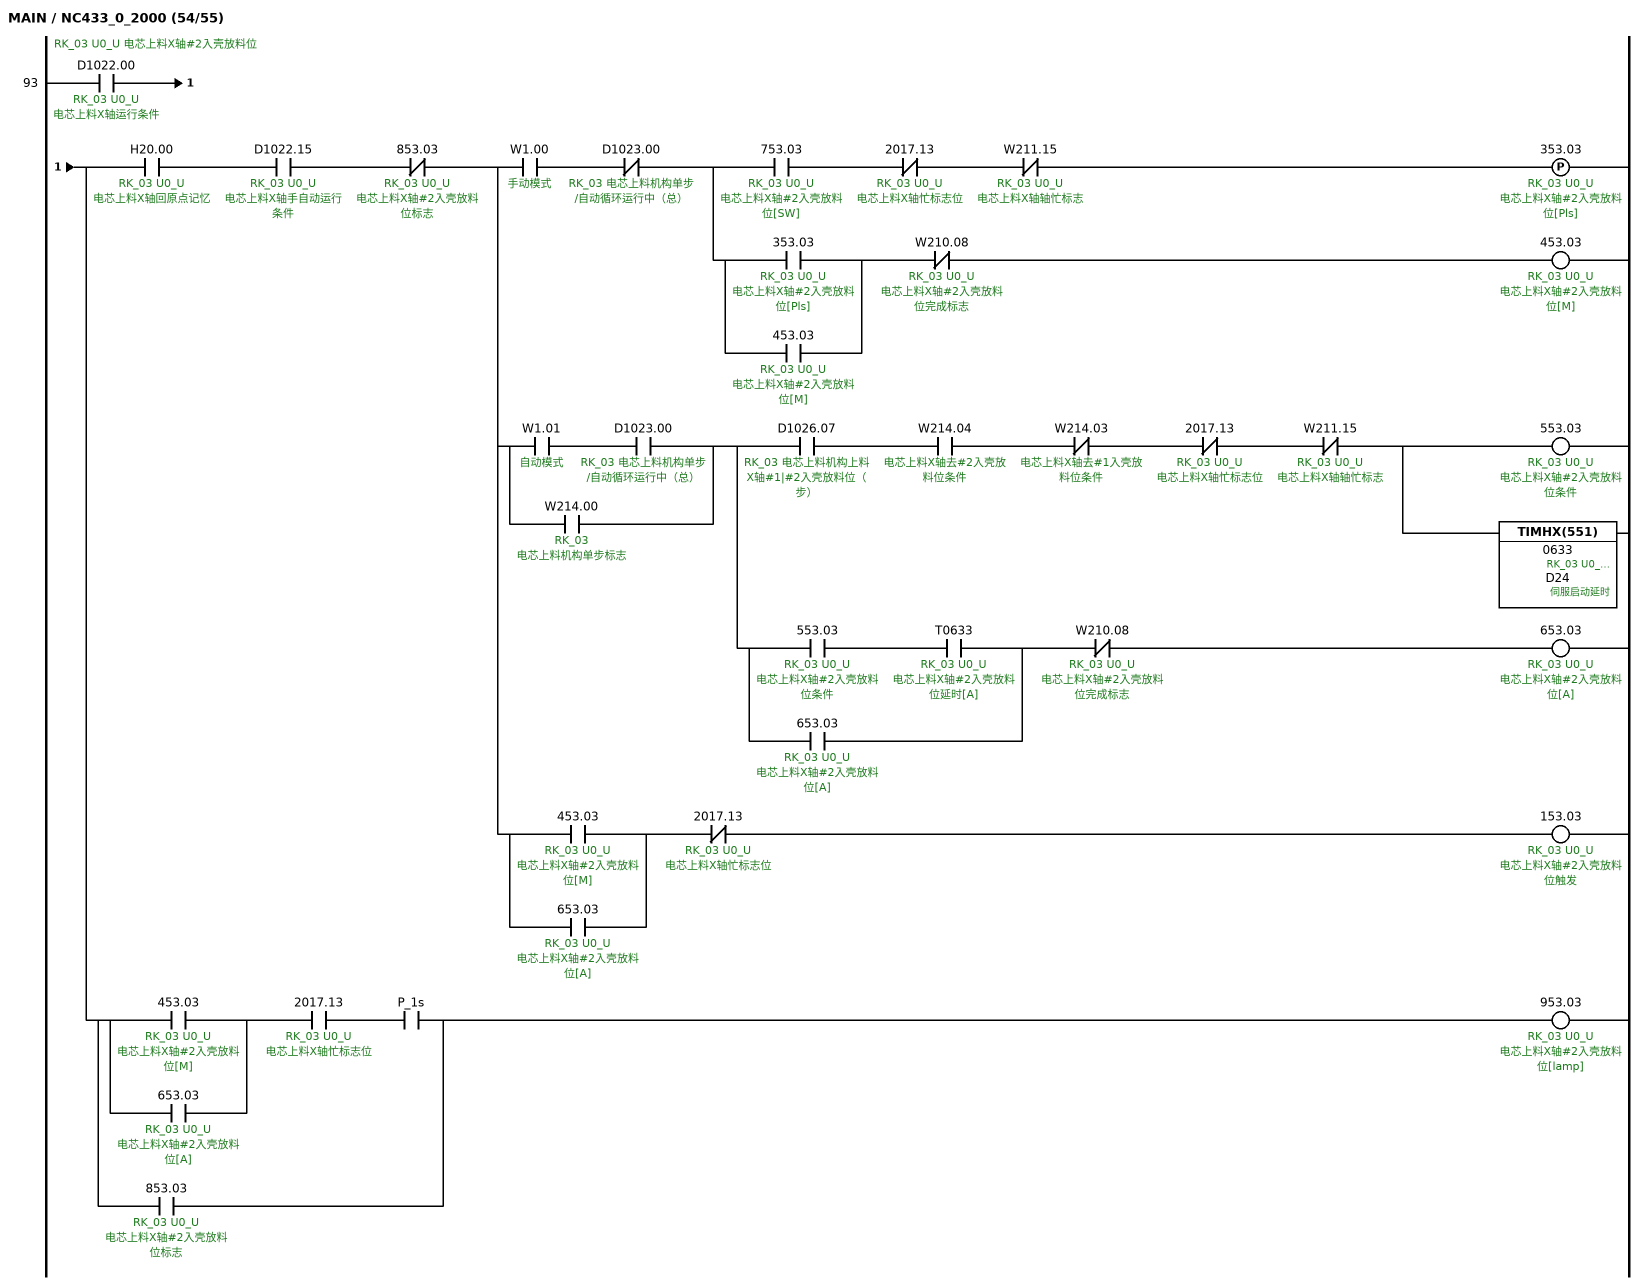
; rung 93: RK_03 U0_U 电芯上料X轴#2入壳放料位
LD D1022.00  ; RK_03 U0_U 电芯上料X轴运行条件
OUT TR0
AND H20.00  ; RK_03 U0_U 电芯上料X轴回原点记忆
AND D1022.15  ; RK_03 U0_U 电芯上料X轴手自动运行条件
ANDNOT 853.03  ; RK_03 U0_U 电芯上料X轴#2入壳放料位标志
OUT TR1
AND W1.00  ; 手动模式
ANDNOT D1023.00  ; RK_03 电芯上料机构单步/自动循环运行中（总）
OUT TR2
AND 753.03  ; RK_03 U0_U 电芯上料X轴#2入壳放料位[SW]
ANDNOT 2017.13  ; RK_03 U0_U 电芯上料X轴忙标志位
ANDNOT W211.15  ; RK_03 U0_U 电芯上料X轴轴忙标志
DIFU(013) 353.03  ; RK_03 U0_U 电芯上料X轴#2入壳放料位[Pls]
LD TR2
LD 353.03  ; RK_03 U0_U 电芯上料X轴#2入壳放料位[Pls]
OR 453.03  ; RK_03 U0_U 电芯上料X轴#2入壳放料位[M]
ANDLD
ANDNOT W210.08  ; RK_03 U0_U 电芯上料X轴#2入壳放料位完成标志
OUT 453.03  ; RK_03 U0_U 电芯上料X轴#2入壳放料位[M]
LD TR1
LD W1.01  ; 自动模式
AND D1023.00  ; RK_03 电芯上料机构单步/自动循环运行中（总）
OR W214.00  ; RK_03  电芯上料机构单步标志
ANDLD
OUT TR2
AND D1026.07  ; RK_03 电芯上料机构上料X轴#1|#2入壳放料位（步）
AND W214.04  ; 电芯上料X轴去#2入壳放料位条件
ANDNOT W214.03  ; 电芯上料X轴去#1入壳放料位条件
ANDNOT 2017.13  ; RK_03 U0_U 电芯上料X轴忙标志位
ANDNOT W211.15  ; RK_03 U0_U 电芯上料X轴轴忙标志
OUT 553.03  ; RK_03 U0_U 电芯上料X轴#2入壳放料位条件
TIMHX(551) 0633 D24  ; 伺服启动延时, RK_03 U0_U 电芯上料X轴#2入壳放料位延时[A]
LD TR2
LD 553.03  ; RK_03 U0_U 电芯上料X轴#2入壳放料位条件
AND T0633  ; RK_03 U0_U 电芯上料X轴#2入壳放料位延时[A]
OR 653.03  ; RK_03 U0_U 电芯上料X轴#2入壳放料位[A]
ANDLD
ANDNOT W210.08  ; RK_03 U0_U 电芯上料X轴#2入壳放料位完成标志
OUT 653.03  ; RK_03 U0_U 电芯上料X轴#2入壳放料位[A]
LD TR1
LD 453.03  ; RK_03 U0_U 电芯上料X轴#2入壳放料位[M]
OR 653.03  ; RK_03 U0_U 电芯上料X轴#2入壳放料位[A]
ANDLD
ANDNOT 2017.13  ; RK_03 U0_U 电芯上料X轴忙标志位
OUT 153.03  ; RK_03 U0_U 电芯上料X轴#2入壳放料位触发
LD TR0
LD 453.03  ; RK_03 U0_U 电芯上料X轴#2入壳放料位[M]
OR 653.03  ; RK_03 U0_U 电芯上料X轴#2入壳放料位[A]
AND 2017.13  ; RK_03 U0_U 电芯上料X轴忙标志位
AND P_1s
OR 853.03  ; RK_03 U0_U 电芯上料X轴#2入壳放料位标志
ANDLD
OUT 953.03  ; RK_03 U0_U 电芯上料X轴#2入壳放料位[lamp]

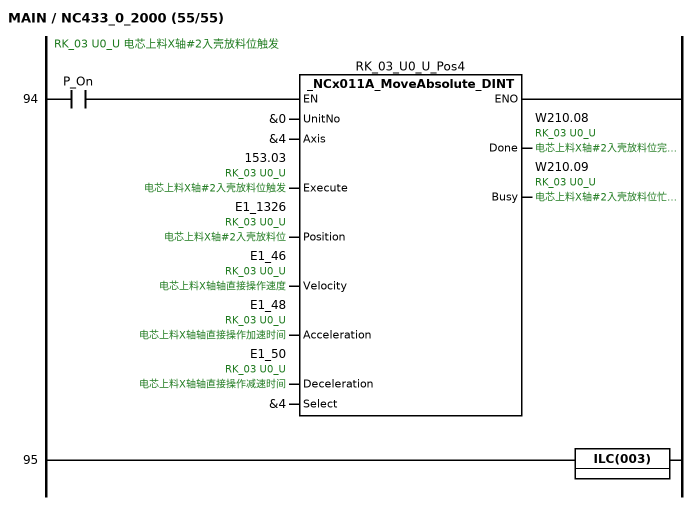
; rung 94: RK_03 U0_U 电芯上料X轴#2入壳放料位触发
LD P_On
CALL RK_03_U0_U_Pos4 : _NCx011A_MoveAbsolute_DINT (UnitNo := &0, Axis := &4, Execute := 153.03, Position := E1_1326, Velocity := E1_46, Acceleration := E1_48, Deceleration := E1_50, Select := &4, Done => W210.08, Busy => W210.09)  ; RK_03 U0_U 电芯上料X轴#2入壳放料位触发, RK_03 U0_U 电芯上料X轴#2入壳放料位, RK_03 U0_U 电芯上料X轴轴直接操作速度, RK_03 U0_U 电芯上料X轴轴直接操作加速时间, RK_03 U0_U 电芯上料X轴轴直接操作减速时间, RK_03 U0_U 电芯上料X轴#2入壳放料位完成标志, RK_03 U0_U 电芯上料X轴#2入壳放料位忙标志
; rung 95
ILC(003)

### Section NC433_2_2020

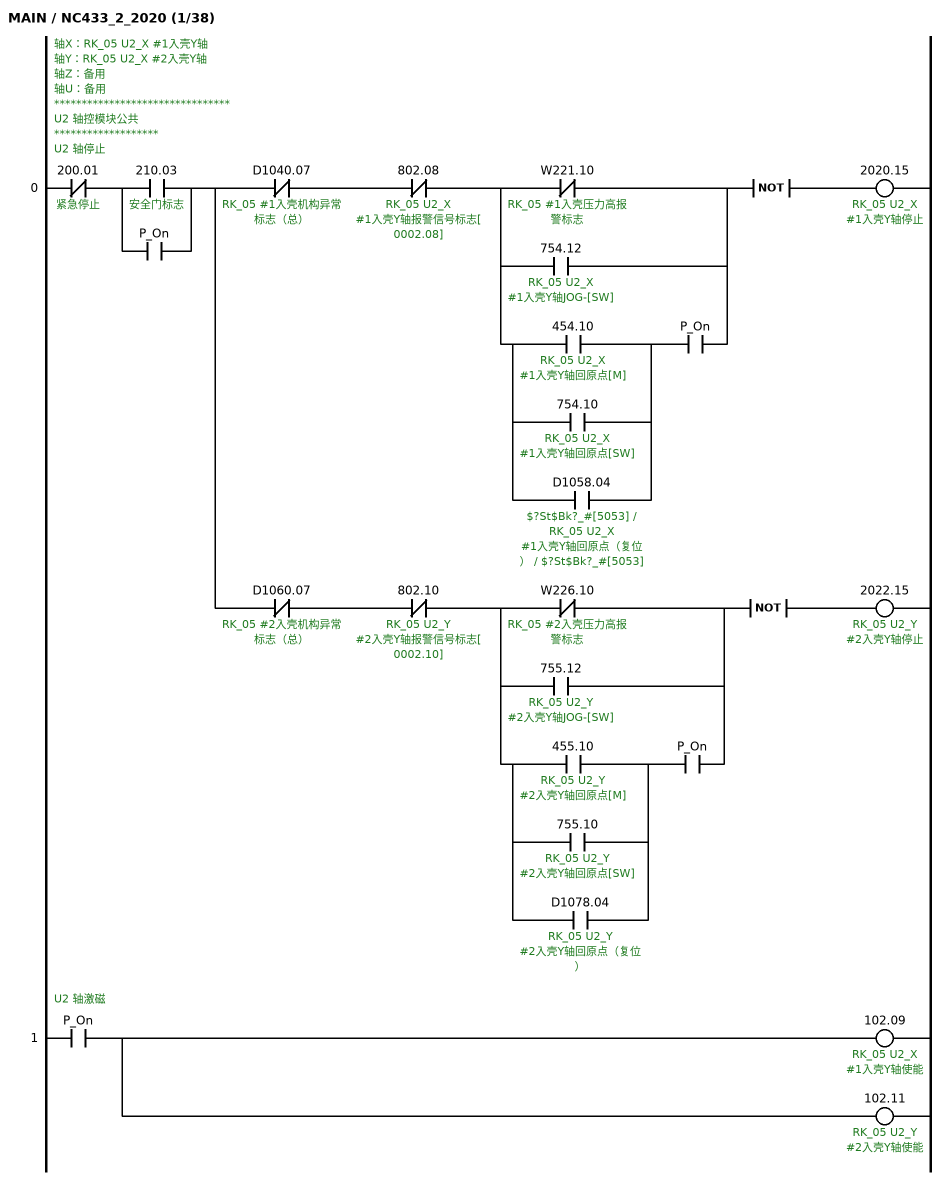
; rung 0: 轴X：RK_05 U2_X #1入壳Y轴 / 轴Y：RK_05 U2_X #2入壳Y轴 / 轴Z：备用 / 轴U：备用 / ******************************** / U2 轴控模块公共 / ******************* / U2 轴停止
LDNOT 200.01  ; 紧急停止
LD 210.03  ; 安全门标志
OR P_On
ANDLD
OUT TR0
ANDNOT D1040.07  ; RK_05 #1入壳机构异常标志（总）
ANDNOT 802.08  ; RK_05 U2_X #1入壳Y轴报警信号标志[0002.08]
LDNOT W221.10  ; RK_05 #1入壳压力高报警标志
OR 754.12  ; RK_05 U2_X #1入壳Y轴JOG-[SW]
LD 454.10  ; RK_05 U2_X #1入壳Y轴回原点[M]
OR 754.10  ; RK_05 U2_X #1入壳Y轴回原点[SW]
OR D1058.04  ; $?St$Bk?_#[5053] / RK_05 U2_X #1入壳Y轴回原点（复位） / $?St$Bk?_#[5053]
AND P_On
ORLD
ANDLD
NOT(520)
OUT 2020.15  ; RK_05 U2_X #1入壳Y轴停止
LD TR0
ANDNOT D1060.07  ; RK_05 #2入壳机构异常标志（总）
ANDNOT 802.10  ; RK_05 U2_Y #2入壳Y轴报警信号标志[0002.10]
LDNOT W226.10  ; RK_05 #2入壳压力高报警标志
OR 755.12  ; RK_05 U2_Y #2入壳Y轴JOG-[SW]
LD 455.10  ; RK_05 U2_Y #2入壳Y轴回原点[M]
OR 755.10  ; RK_05 U2_Y #2入壳Y轴回原点[SW]
OR D1078.04  ; RK_05 U2_Y #2入壳Y轴回原点（复位）
AND P_On
ORLD
ANDLD
NOT(520)
OUT 2022.15  ; RK_05 U2_Y #2入壳Y轴停止
; rung 1: U2 轴激磁
LD P_On
OUT 102.09  ; RK_05 U2_X #1入壳Y轴使能
OUT 102.11  ; RK_05 U2_Y #2入壳Y轴使能

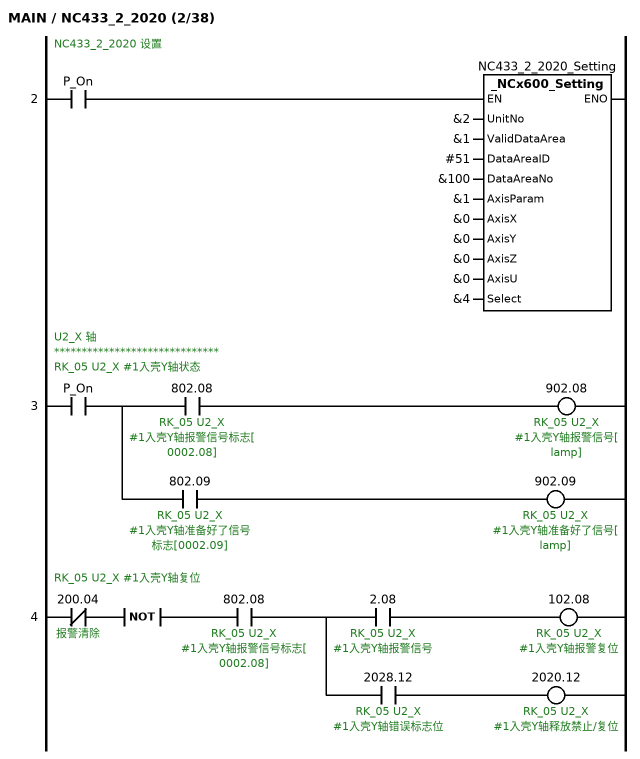
; rung 2: NC433_2_2020 设置
LD P_On
CALL NC433_2_2020_Setting : _NCx600_Setting (UnitNo := &2, ValidDataArea := &1, DataAreaID := #51, DataAreaNo := &100, AxisParam := &1, AxisX := &0, AxisY := &0, AxisZ := &0, AxisU := &0, Select := &4)
; rung 3: U2_X 轴 / ****************************** / RK_05 U2_X #1入壳Y轴状态
LD P_On
OUT TR0
AND 802.08  ; RK_05 U2_X #1入壳Y轴报警信号标志[0002.08]
OUT 902.08  ; RK_05 U2_X #1入壳Y轴报警信号[lamp]
LD TR0
AND 802.09  ; RK_05 U2_X #1入壳Y轴准备好了信号标志[0002.09]
OUT 902.09  ; RK_05 U2_X #1入壳Y轴准备好了信号[lamp]
; rung 4: RK_05 U2_X #1入壳Y轴复位
LDNOT 200.04  ; 报警清除
NOT(520)
AND 802.08  ; RK_05 U2_X #1入壳Y轴报警信号标志[0002.08]
OUT TR0
AND 2.08  ; RK_05 U2_X #1入壳Y轴报警信号
OUT 102.08  ; RK_05 U2_X #1入壳Y轴报警复位
LD TR0
AND 2028.12  ; RK_05 U2_X #1入壳Y轴错误标志位
OUT 2020.12  ; RK_05 U2_X #1入壳Y轴释放禁止/复位

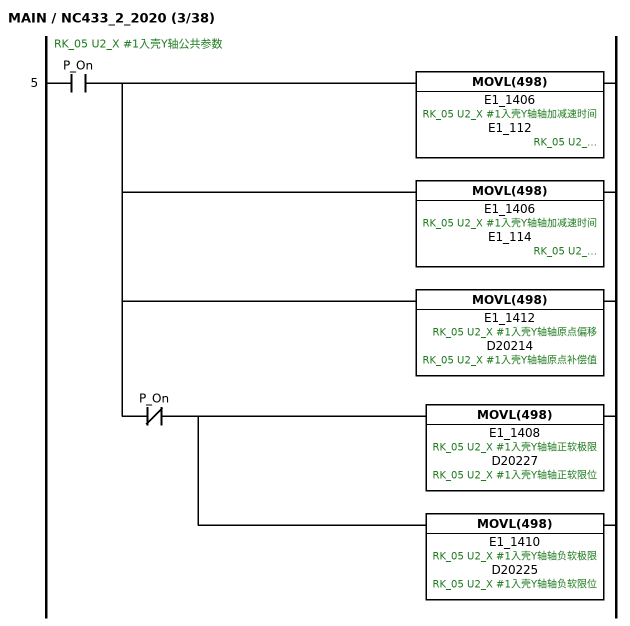
; rung 5: RK_05 U2_X #1入壳Y轴公共参数
LD P_On
MOVL(498) E1_1406 E1_112  ; RK_05 U2_X #1入壳Y轴轴加减速时间, RK_05 U2_X #1入壳Y轴轴直接操作加速时间
MOVL(498) E1_1406 E1_114  ; RK_05 U2_X #1入壳Y轴轴加减速时间, RK_05 U2_X #1入壳Y轴轴直接操作减速时间
MOVL(498) E1_1412 D20214  ; RK_05 U2_X #1入壳Y轴轴原点偏移, RK_05 U2_X #1入壳Y轴轴原点补偿值
ANDNOT P_On
MOVL(498) E1_1408 D20227  ; RK_05 U2_X #1入壳Y轴轴正软极限, RK_05 U2_X #1入壳Y轴轴正软限位
MOVL(498) E1_1410 D20225  ; RK_05 U2_X #1入壳Y轴轴负软极限, RK_05 U2_X #1入壳Y轴轴负软限位

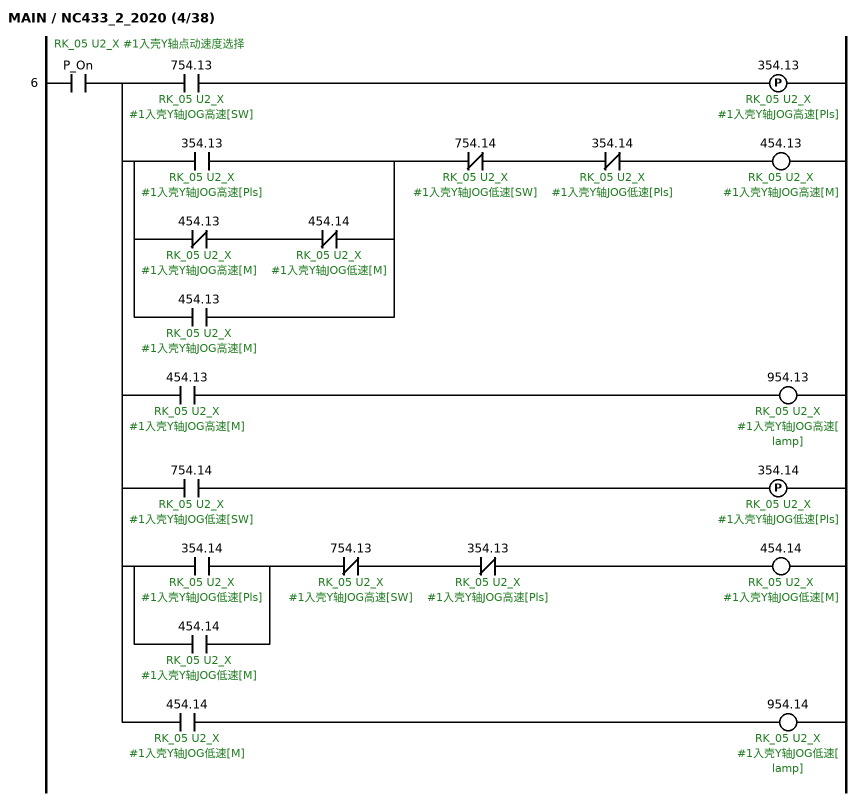
; rung 6: RK_05 U2_X #1入壳Y轴点动速度选择
LD P_On
OUT TR0
AND 754.13  ; RK_05 U2_X #1入壳Y轴JOG高速[SW]
DIFU(013) 354.13  ; RK_05 U2_X #1入壳Y轴JOG高速[Pls]
LD TR0
LD 354.13  ; RK_05 U2_X #1入壳Y轴JOG高速[Pls]
LDNOT 454.13  ; RK_05 U2_X #1入壳Y轴JOG高速[M]
ANDNOT 454.14  ; RK_05 U2_X #1入壳Y轴JOG低速[M]
ORLD
OR 454.13  ; RK_05 U2_X #1入壳Y轴JOG高速[M]
ANDLD
ANDNOT 754.14  ; RK_05 U2_X #1入壳Y轴JOG低速[SW]
ANDNOT 354.14  ; RK_05 U2_X #1入壳Y轴JOG低速[Pls]
OUT 454.13  ; RK_05 U2_X #1入壳Y轴JOG高速[M]
LD TR0
AND 454.13  ; RK_05 U2_X #1入壳Y轴JOG高速[M]
OUT 954.13  ; RK_05 U2_X #1入壳Y轴JOG高速[lamp]
LD TR0
AND 754.14  ; RK_05 U2_X #1入壳Y轴JOG低速[SW]
DIFU(013) 354.14  ; RK_05 U2_X #1入壳Y轴JOG低速[Pls]
LD TR0
LD 354.14  ; RK_05 U2_X #1入壳Y轴JOG低速[Pls]
OR 454.14  ; RK_05 U2_X #1入壳Y轴JOG低速[M]
ANDLD
ANDNOT 754.13  ; RK_05 U2_X #1入壳Y轴JOG高速[SW]
ANDNOT 354.13  ; RK_05 U2_X #1入壳Y轴JOG高速[Pls]
OUT 454.14  ; RK_05 U2_X #1入壳Y轴JOG低速[M]
LD TR0
AND 454.14  ; RK_05 U2_X #1入壳Y轴JOG低速[M]
OUT 954.14  ; RK_05 U2_X #1入壳Y轴JOG低速[lamp]

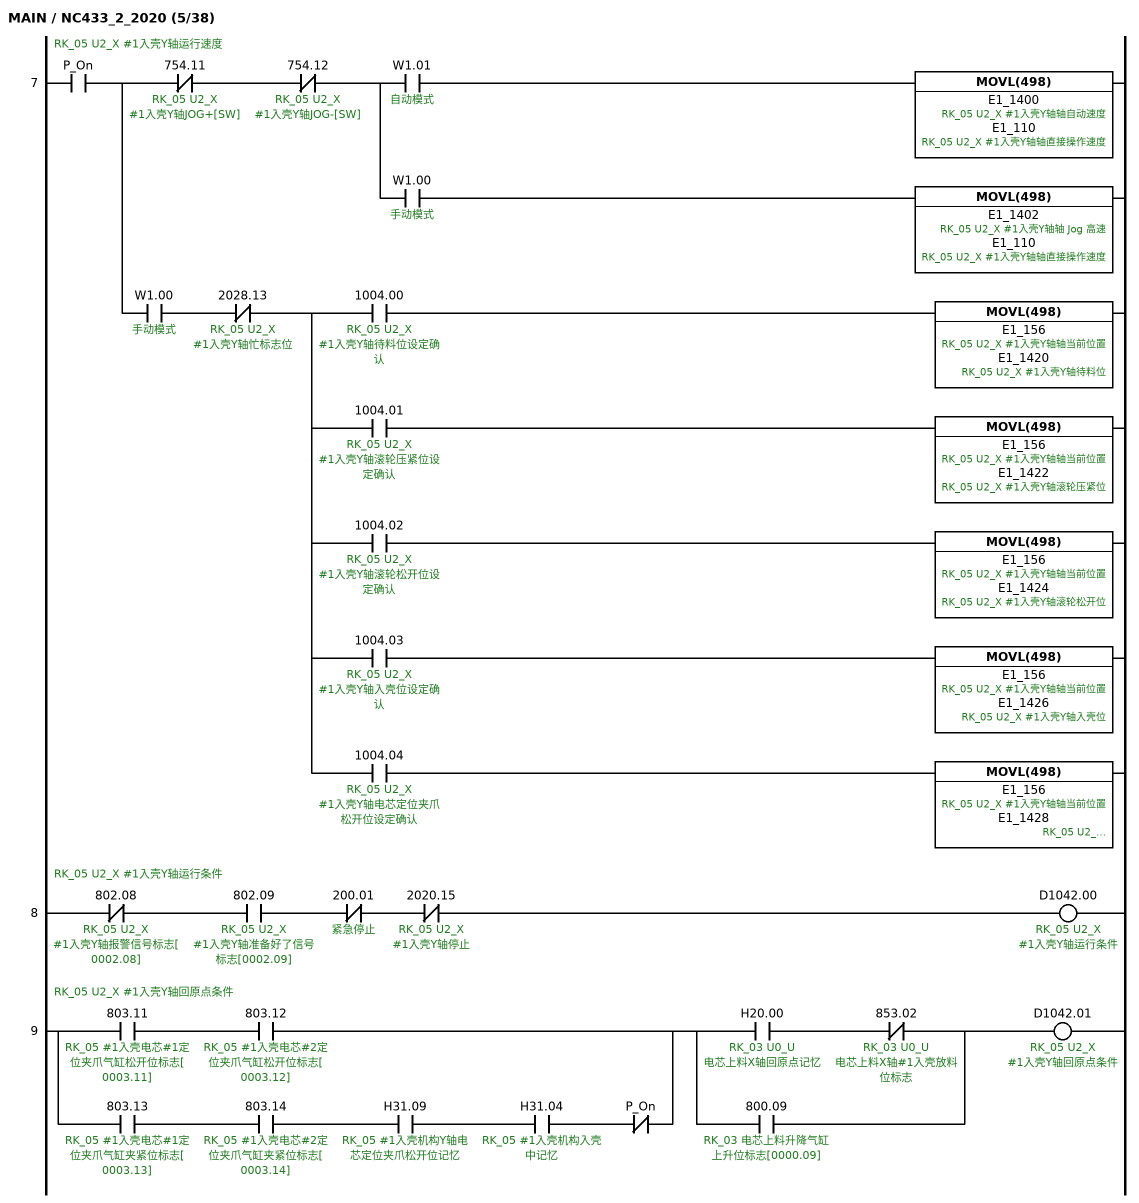
; rung 7: RK_05 U2_X #1入壳Y轴运行速度
LD P_On
OUT TR0
ANDNOT 754.11  ; RK_05 U2_X #1入壳Y轴JOG+[SW]
ANDNOT 754.12  ; RK_05 U2_X #1入壳Y轴JOG-[SW]
OUT TR1
AND W1.01  ; 自动模式
MOVL(498) E1_1400 E1_110  ; RK_05 U2_X #1入壳Y轴轴自动速度, RK_05 U2_X #1入壳Y轴轴直接操作速度
LD TR1
AND W1.00  ; 手动模式
MOVL(498) E1_1402 E1_110  ; RK_05 U2_X #1入壳Y轴轴 Jog 高速, RK_05 U2_X #1入壳Y轴轴直接操作速度
LD TR0
AND W1.00  ; 手动模式
ANDNOT 2028.13  ; RK_05 U2_X #1入壳Y轴忙标志位
OUT TR0
AND 1004.00  ; RK_05 U2_X #1入壳Y轴待料位设定确认
MOVL(498) E1_156 E1_1420  ; RK_05 U2_X #1入壳Y轴轴当前位置, RK_05 U2_X #1入壳Y轴待料位
LD TR0
AND 1004.01  ; RK_05 U2_X #1入壳Y轴滚轮压紧位设定确认
MOVL(498) E1_156 E1_1422  ; RK_05 U2_X #1入壳Y轴轴当前位置, RK_05 U2_X #1入壳Y轴滚轮压紧位
LD TR0
AND 1004.02  ; RK_05 U2_X #1入壳Y轴滚轮松开位设定确认
MOVL(498) E1_156 E1_1424  ; RK_05 U2_X #1入壳Y轴轴当前位置, RK_05 U2_X #1入壳Y轴滚轮松开位
LD TR0
AND 1004.03  ; RK_05 U2_X #1入壳Y轴入壳位设定确认
MOVL(498) E1_156 E1_1426  ; RK_05 U2_X #1入壳Y轴轴当前位置, RK_05 U2_X #1入壳Y轴入壳位
LD TR0
AND 1004.04  ; RK_05 U2_X #1入壳Y轴电芯定位夹爪松开位设定确认
MOVL(498) E1_156 E1_1428  ; RK_05 U2_X #1入壳Y轴轴当前位置, RK_05 U2_X #1入壳Y轴电芯定位夹爪松开位
; rung 8: RK_05 U2_X #1入壳Y轴运行条件
LDNOT 802.08  ; RK_05 U2_X #1入壳Y轴报警信号标志[0002.08]
AND 802.09  ; RK_05 U2_X #1入壳Y轴准备好了信号标志[0002.09]
ANDNOT 200.01  ; 紧急停止
ANDNOT 2020.15  ; RK_05 U2_X #1入壳Y轴停止
OUT D1042.00  ; RK_05 U2_X #1入壳Y轴运行条件
; rung 9: RK_05 U2_X #1入壳Y轴回原点条件
LD 803.11  ; RK_05 #1入壳电芯#1定位夹爪气缸松开位标志[0003.11]
AND 803.12  ; RK_05 #1入壳电芯#2定位夹爪气缸松开位标志[0003.12]
LD 803.13  ; RK_05 #1入壳电芯#1定位夹爪气缸夹紧位标志[0003.13]
AND 803.14  ; RK_05 #1入壳电芯#2定位夹爪气缸夹紧位标志[0003.14]
AND H31.09  ; RK_05 #1入壳机构Y轴电芯定位夹爪松开位记忆
AND H31.04  ; RK_05 #1入壳机构入壳中记忆
ANDNOT P_On
ORLD
LD H20.00  ; RK_03 U0_U 电芯上料X轴回原点记忆
ANDNOT 853.02  ; RK_03 U0_U 电芯上料X轴#1入壳放料位标志
OR 800.09  ; RK_03 电芯上料升降气缸上升位标志[0000.09]
ANDLD
OUT D1042.01  ; RK_05 U2_X #1入壳Y轴回原点条件

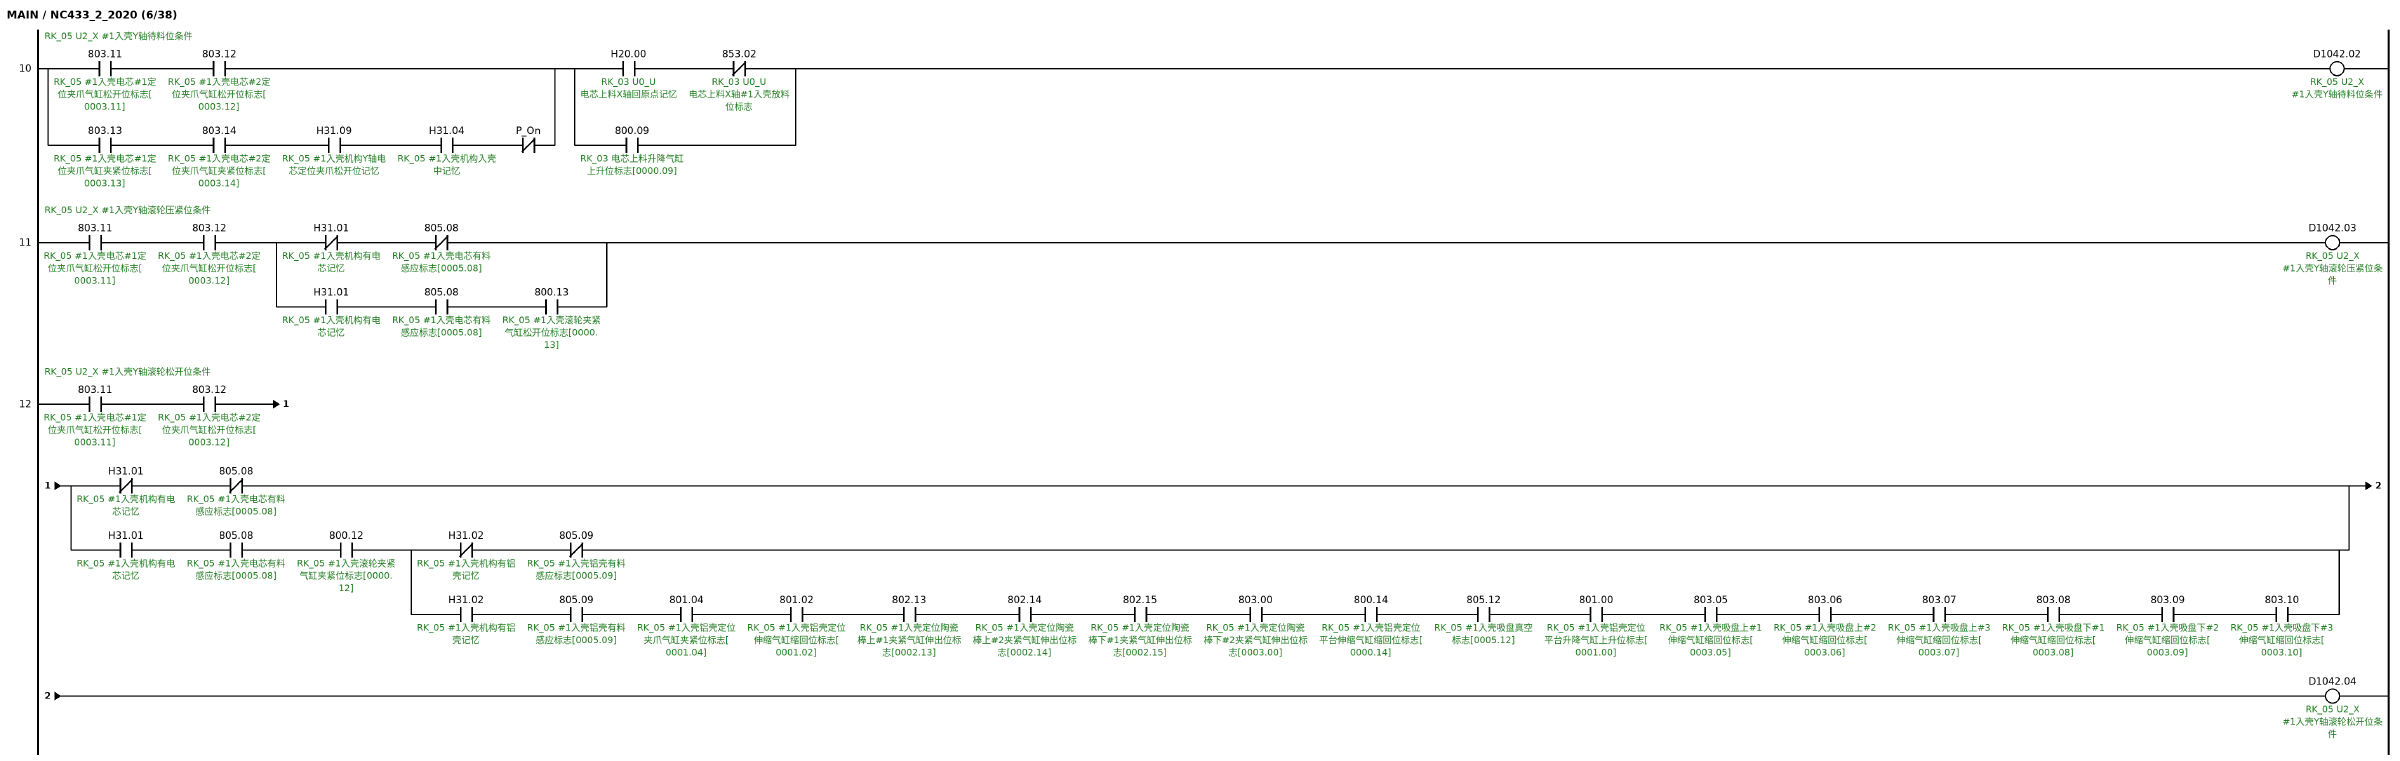
; rung 10: RK_05 U2_X #1入壳Y轴待料位条件
LD 803.11  ; RK_05 #1入壳电芯#1定位夹爪气缸松开位标志[0003.11]
AND 803.12  ; RK_05 #1入壳电芯#2定位夹爪气缸松开位标志[0003.12]
LD 803.13  ; RK_05 #1入壳电芯#1定位夹爪气缸夹紧位标志[0003.13]
AND 803.14  ; RK_05 #1入壳电芯#2定位夹爪气缸夹紧位标志[0003.14]
AND H31.09  ; RK_05 #1入壳机构Y轴电芯定位夹爪松开位记忆
AND H31.04  ; RK_05 #1入壳机构入壳中记忆
ANDNOT P_On
ORLD
LD H20.00  ; RK_03 U0_U 电芯上料X轴回原点记忆
ANDNOT 853.02  ; RK_03 U0_U 电芯上料X轴#1入壳放料位标志
OR 800.09  ; RK_03 电芯上料升降气缸上升位标志[0000.09]
ANDLD
OUT D1042.02  ; RK_05 U2_X #1入壳Y轴待料位条件
; rung 11: RK_05 U2_X #1入壳Y轴滚轮压紧位条件
LD 803.11  ; RK_05 #1入壳电芯#1定位夹爪气缸松开位标志[0003.11]
AND 803.12  ; RK_05 #1入壳电芯#2定位夹爪气缸松开位标志[0003.12]
LDNOT H31.01  ; RK_05 #1入壳机构有电芯记忆
ANDNOT 805.08  ; RK_05 #1入壳电芯有料感应标志[0005.08]
LD H31.01  ; RK_05 #1入壳机构有电芯记忆
AND 805.08  ; RK_05 #1入壳电芯有料感应标志[0005.08]
AND 800.13  ; RK_05 #1入壳滚轮夹紧气缸松开位标志[0000.13]
ORLD
ANDLD
OUT D1042.03  ; RK_05 U2_X #1入壳Y轴滚轮压紧位条件
; rung 12: RK_05 U2_X #1入壳Y轴滚轮松开位条件
LD 803.11  ; RK_05 #1入壳电芯#1定位夹爪气缸松开位标志[0003.11]
AND 803.12  ; RK_05 #1入壳电芯#2定位夹爪气缸松开位标志[0003.12]
LDNOT H31.01  ; RK_05 #1入壳机构有电芯记忆
ANDNOT 805.08  ; RK_05 #1入壳电芯有料感应标志[0005.08]
LD H31.01  ; RK_05 #1入壳机构有电芯记忆
AND 805.08  ; RK_05 #1入壳电芯有料感应标志[0005.08]
AND 800.12  ; RK_05 #1入壳滚轮夹紧气缸夹紧位标志[0000.12]
LDNOT H31.02  ; RK_05 #1入壳机构有铝壳记忆
ANDNOT 805.09  ; RK_05 #1入壳铝壳有料感应标志[0005.09]
LD H31.02  ; RK_05 #1入壳机构有铝壳记忆
AND 805.09  ; RK_05 #1入壳铝壳有料感应标志[0005.09]
AND 801.04  ; RK_05 #1入壳铝壳定位夹爪气缸夹紧位标志[0001.04]
AND 801.02  ; RK_05 #1入壳铝壳定位伸缩气缸缩回位标志[0001.02]
AND 802.13  ; RK_05 #1入壳定位陶瓷棒上#1夹紧气缸伸出位标志[0002.13]
AND 802.14  ; RK_05 #1入壳定位陶瓷棒上#2夹紧气缸伸出位标志[0002.14]
AND 802.15  ; RK_05 #1入壳定位陶瓷棒下#1夹紧气缸伸出位标志[0002.15]
AND 803.00  ; RK_05 #1入壳定位陶瓷棒下#2夹紧气缸伸出位标志[0003.00]
AND 800.14  ; RK_05 #1入壳铝壳定位平台伸缩气缸缩回位标志[0000.14]
AND 805.12  ; RK_05 #1入壳吸盘真空标志[0005.12]
AND 801.00  ; RK_05 #1入壳铝壳定位平台升降气缸上升位标志[0001.00]
AND 803.05  ; RK_05 #1入壳吸盘上#1伸缩气缸缩回位标志[0003.05]
AND 803.06  ; RK_05 #1入壳吸盘上#2伸缩气缸缩回位标志[0003.06]
AND 803.07  ; RK_05 #1入壳吸盘上#3伸缩气缸缩回位标志[0003.07]
AND 803.08  ; RK_05 #1入壳吸盘下#1伸缩气缸缩回位标志[0003.08]
AND 803.09  ; RK_05 #1入壳吸盘下#2伸缩气缸缩回位标志[0003.09]
AND 803.10  ; RK_05 #1入壳吸盘下#3伸缩气缸缩回位标志[0003.10]
ORLD
ANDLD
ORLD
ANDLD
OUT D1042.04  ; RK_05 U2_X #1入壳Y轴滚轮松开位条件

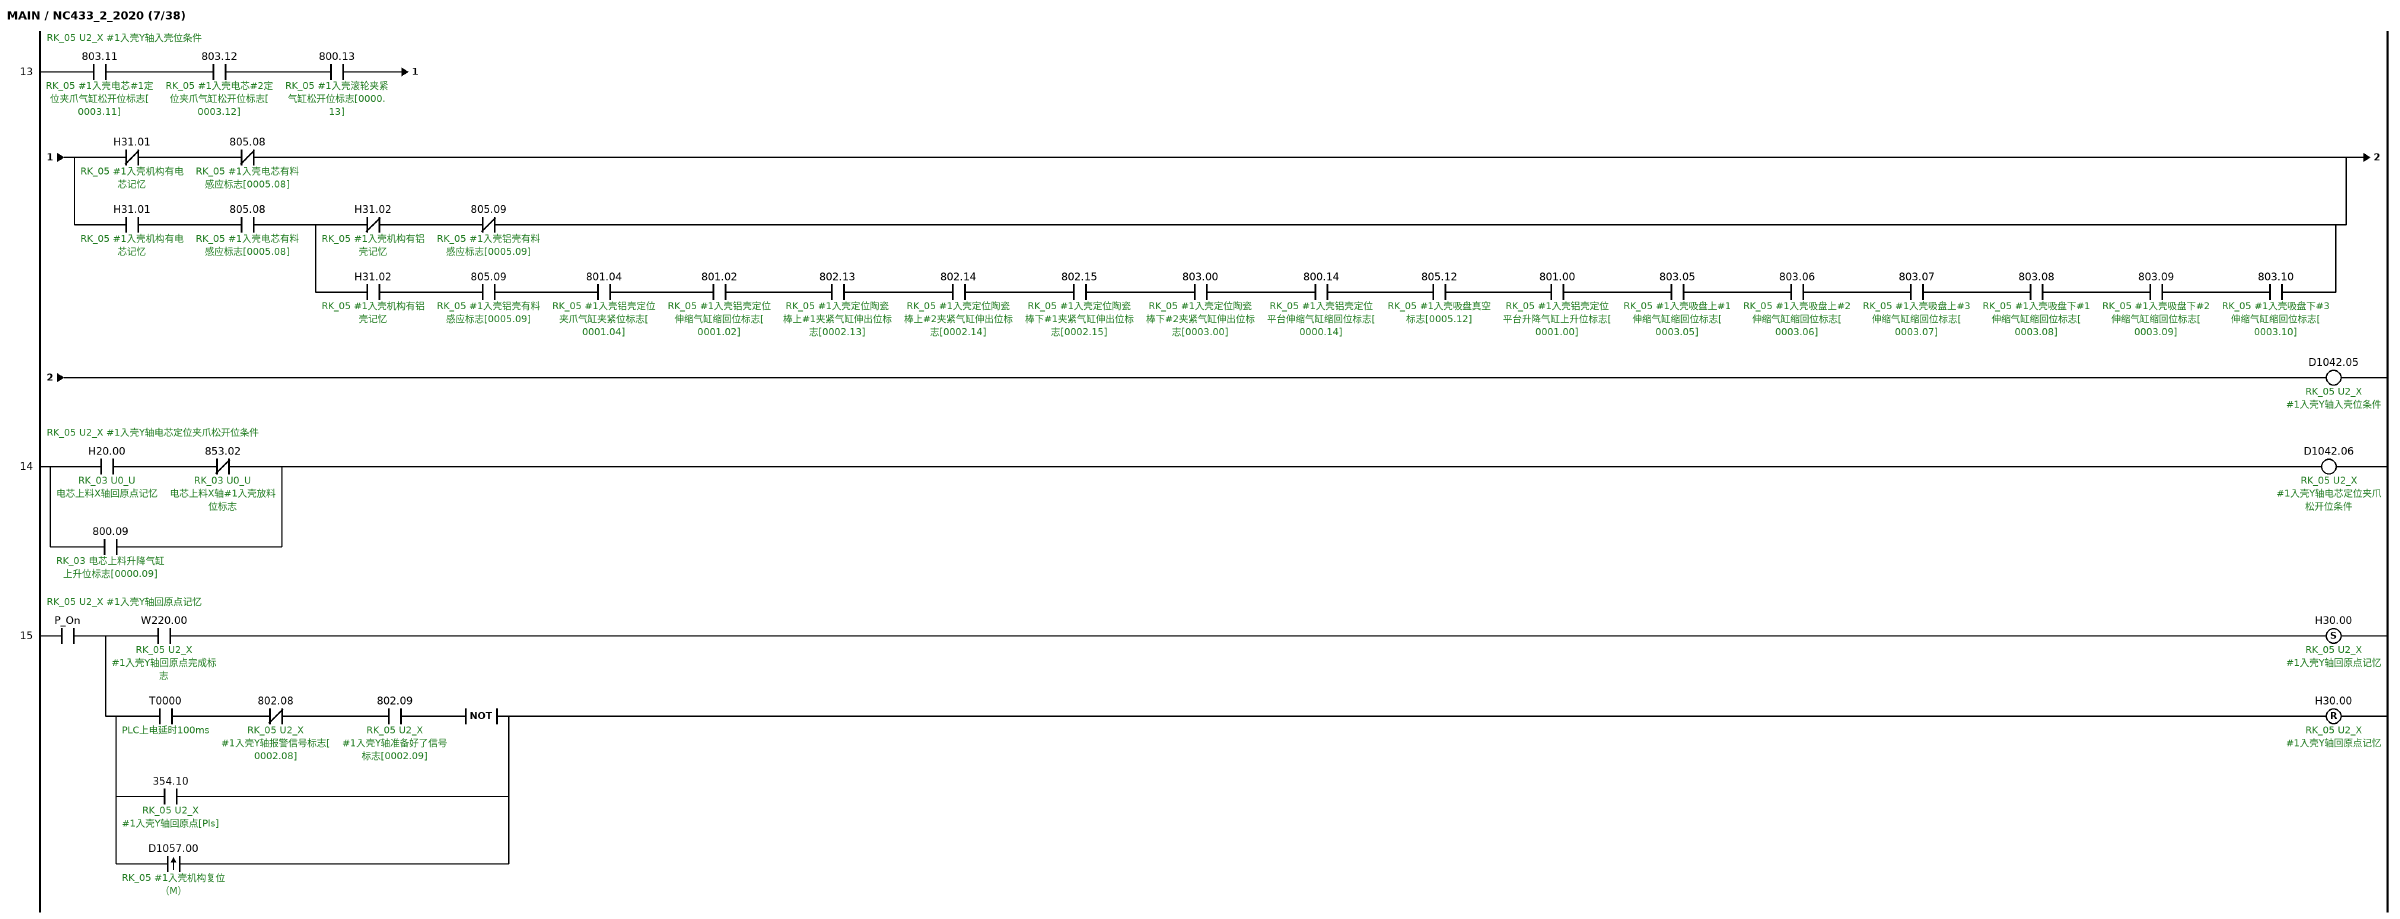
; rung 13: RK_05 U2_X #1入壳Y轴入壳位条件
LD 803.11  ; RK_05 #1入壳电芯#1定位夹爪气缸松开位标志[0003.11]
AND 803.12  ; RK_05 #1入壳电芯#2定位夹爪气缸松开位标志[0003.12]
AND 800.13  ; RK_05 #1入壳滚轮夹紧气缸松开位标志[0000.13]
LDNOT H31.01  ; RK_05 #1入壳机构有电芯记忆
ANDNOT 805.08  ; RK_05 #1入壳电芯有料感应标志[0005.08]
LD H31.01  ; RK_05 #1入壳机构有电芯记忆
AND 805.08  ; RK_05 #1入壳电芯有料感应标志[0005.08]
LDNOT H31.02  ; RK_05 #1入壳机构有铝壳记忆
ANDNOT 805.09  ; RK_05 #1入壳铝壳有料感应标志[0005.09]
LD H31.02  ; RK_05 #1入壳机构有铝壳记忆
AND 805.09  ; RK_05 #1入壳铝壳有料感应标志[0005.09]
AND 801.04  ; RK_05 #1入壳铝壳定位夹爪气缸夹紧位标志[0001.04]
AND 801.02  ; RK_05 #1入壳铝壳定位伸缩气缸缩回位标志[0001.02]
AND 802.13  ; RK_05 #1入壳定位陶瓷棒上#1夹紧气缸伸出位标志[0002.13]
AND 802.14  ; RK_05 #1入壳定位陶瓷棒上#2夹紧气缸伸出位标志[0002.14]
AND 802.15  ; RK_05 #1入壳定位陶瓷棒下#1夹紧气缸伸出位标志[0002.15]
AND 803.00  ; RK_05 #1入壳定位陶瓷棒下#2夹紧气缸伸出位标志[0003.00]
AND 800.14  ; RK_05 #1入壳铝壳定位平台伸缩气缸缩回位标志[0000.14]
AND 805.12  ; RK_05 #1入壳吸盘真空标志[0005.12]
AND 801.00  ; RK_05 #1入壳铝壳定位平台升降气缸上升位标志[0001.00]
AND 803.05  ; RK_05 #1入壳吸盘上#1伸缩气缸缩回位标志[0003.05]
AND 803.06  ; RK_05 #1入壳吸盘上#2伸缩气缸缩回位标志[0003.06]
AND 803.07  ; RK_05 #1入壳吸盘上#3伸缩气缸缩回位标志[0003.07]
AND 803.08  ; RK_05 #1入壳吸盘下#1伸缩气缸缩回位标志[0003.08]
AND 803.09  ; RK_05 #1入壳吸盘下#2伸缩气缸缩回位标志[0003.09]
AND 803.10  ; RK_05 #1入壳吸盘下#3伸缩气缸缩回位标志[0003.10]
ORLD
ANDLD
ORLD
ANDLD
OUT D1042.05  ; RK_05 U2_X #1入壳Y轴入壳位条件
; rung 14: RK_05 U2_X #1入壳Y轴电芯定位夹爪松开位条件
LD H20.00  ; RK_03 U0_U 电芯上料X轴回原点记忆
ANDNOT 853.02  ; RK_03 U0_U 电芯上料X轴#1入壳放料位标志
OR 800.09  ; RK_03 电芯上料升降气缸上升位标志[0000.09]
OUT D1042.06  ; RK_05 U2_X #1入壳Y轴电芯定位夹爪松开位条件
; rung 15: RK_05 U2_X #1入壳Y轴回原点记忆
LD P_On
OUT TR0
AND W220.00  ; RK_05 U2_X #1入壳Y轴回原点完成标志
SET H30.00  ; RK_05 U2_X #1入壳Y轴回原点记忆
LD TR0
LD T0000  ; PLC上电延时100ms
ANDNOT 802.08  ; RK_05 U2_X #1入壳Y轴报警信号标志[0002.08]
AND 802.09  ; RK_05 U2_X #1入壳Y轴准备好了信号标志[0002.09]
NOT(520)
OR 354.10  ; RK_05 U2_X #1入壳Y轴回原点[Pls]
@OR D1057.00  ; RK_05 #1入壳机构复位（M）
ANDLD
RSET H30.00  ; RK_05 U2_X #1入壳Y轴回原点记忆

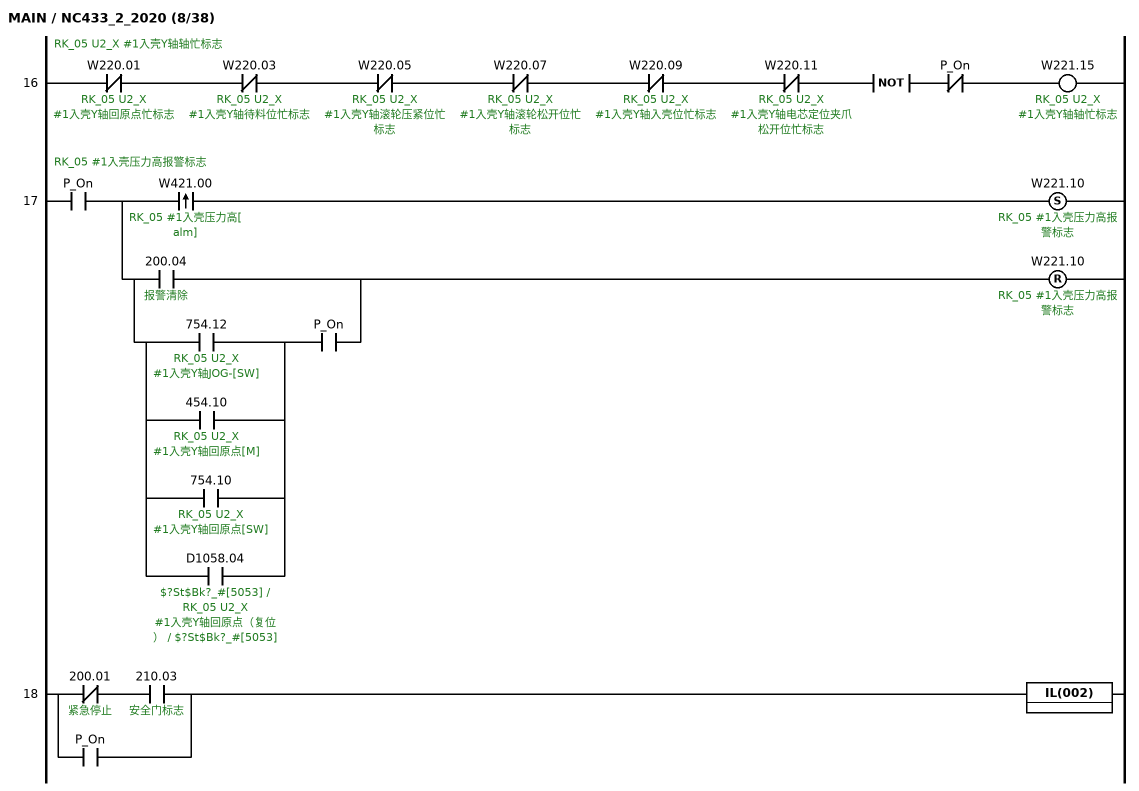
; rung 16: RK_05 U2_X #1入壳Y轴轴忙标志
LDNOT W220.01  ; RK_05 U2_X #1入壳Y轴回原点忙标志
ANDNOT W220.03  ; RK_05 U2_X #1入壳Y轴待料位忙标志
ANDNOT W220.05  ; RK_05 U2_X #1入壳Y轴滚轮压紧位忙标志
ANDNOT W220.07  ; RK_05 U2_X #1入壳Y轴滚轮松开位忙标志
ANDNOT W220.09  ; RK_05 U2_X #1入壳Y轴入壳位忙标志
ANDNOT W220.11  ; RK_05 U2_X #1入壳Y轴电芯定位夹爪松开位忙标志
NOT(520)
ANDNOT P_On
OUT W221.15  ; RK_05 U2_X #1入壳Y轴轴忙标志
; rung 17: RK_05 #1入壳压力高报警标志
LD P_On
OUT TR0
@AND W421.00  ; RK_05 #1入壳压力高[alm]
SET W221.10  ; RK_05 #1入壳压力高报警标志
LD TR0
LD 200.04  ; 报警清除
LD 754.12  ; RK_05 U2_X #1入壳Y轴JOG-[SW]
OR 454.10  ; RK_05 U2_X #1入壳Y轴回原点[M]
OR 754.10  ; RK_05 U2_X #1入壳Y轴回原点[SW]
OR D1058.04  ; $?St$Bk?_#[5053] / RK_05 U2_X #1入壳Y轴回原点（复位） / $?St$Bk?_#[5053]
AND P_On
ORLD
ANDLD
RSET W221.10  ; RK_05 #1入壳压力高报警标志
; rung 18
LDNOT 200.01  ; 紧急停止
AND 210.03  ; 安全门标志
OR P_On
IL(002)

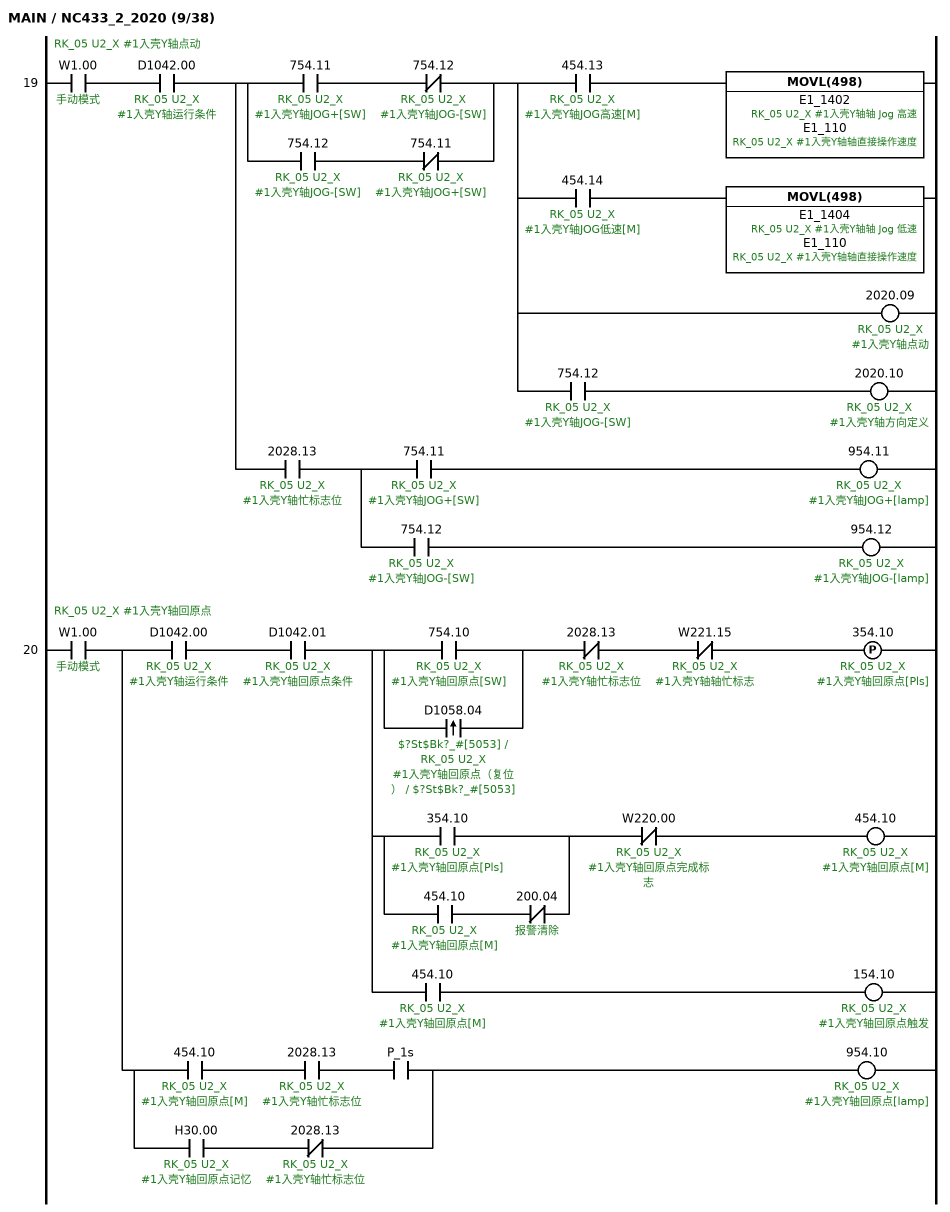
; rung 19: RK_05 U2_X #1入壳Y轴点动
LD W1.00  ; 手动模式
AND D1042.00  ; RK_05 U2_X #1入壳Y轴运行条件
OUT TR0
LD 754.11  ; RK_05 U2_X #1入壳Y轴JOG+[SW]
ANDNOT 754.12  ; RK_05 U2_X #1入壳Y轴JOG-[SW]
LD 754.12  ; RK_05 U2_X #1入壳Y轴JOG-[SW]
ANDNOT 754.11  ; RK_05 U2_X #1入壳Y轴JOG+[SW]
ORLD
ANDLD
OUT TR1
AND 454.13  ; RK_05 U2_X #1入壳Y轴JOG高速[M]
MOVL(498) E1_1402 E1_110  ; RK_05 U2_X #1入壳Y轴轴 Jog 高速, RK_05 U2_X #1入壳Y轴轴直接操作速度
LD TR1
AND 454.14  ; RK_05 U2_X #1入壳Y轴JOG低速[M]
MOVL(498) E1_1404 E1_110  ; RK_05 U2_X #1入壳Y轴轴 Jog 低速, RK_05 U2_X #1入壳Y轴轴直接操作速度
LD TR1
OUT 2020.09  ; RK_05 U2_X #1入壳Y轴点动
AND 754.12  ; RK_05 U2_X #1入壳Y轴JOG-[SW]
OUT 2020.10  ; RK_05 U2_X #1入壳Y轴方向定义
LD TR0
AND 2028.13  ; RK_05 U2_X #1入壳Y轴忙标志位
OUT TR0
AND 754.11  ; RK_05 U2_X #1入壳Y轴JOG+[SW]
OUT 954.11  ; RK_05 U2_X #1入壳Y轴JOG+[lamp]
LD TR0
AND 754.12  ; RK_05 U2_X #1入壳Y轴JOG-[SW]
OUT 954.12  ; RK_05 U2_X #1入壳Y轴JOG-[lamp]
; rung 20: RK_05 U2_X #1入壳Y轴回原点
LD W1.00  ; 手动模式
OUT TR0
AND D1042.00  ; RK_05 U2_X #1入壳Y轴运行条件
AND D1042.01  ; RK_05 U2_X #1入壳Y轴回原点条件
OUT TR1
LD 754.10  ; RK_05 U2_X #1入壳Y轴回原点[SW]
@OR D1058.04  ; $?St$Bk?_#[5053] / RK_05 U2_X #1入壳Y轴回原点（复位） / $?St$Bk?_#[5053]
ANDLD
ANDNOT 2028.13  ; RK_05 U2_X #1入壳Y轴忙标志位
ANDNOT W221.15  ; RK_05 U2_X #1入壳Y轴轴忙标志
DIFU(013) 354.10  ; RK_05 U2_X #1入壳Y轴回原点[Pls]
LD TR1
LD 354.10  ; RK_05 U2_X #1入壳Y轴回原点[Pls]
LD 454.10  ; RK_05 U2_X #1入壳Y轴回原点[M]
ANDNOT 200.04  ; 报警清除
ORLD
ANDLD
ANDNOT W220.00  ; RK_05 U2_X #1入壳Y轴回原点完成标志
OUT 454.10  ; RK_05 U2_X #1入壳Y轴回原点[M]
LD TR1
AND 454.10  ; RK_05 U2_X #1入壳Y轴回原点[M]
OUT 154.10  ; RK_05 U2_X #1入壳Y轴回原点触发
LD TR0
LD 454.10  ; RK_05 U2_X #1入壳Y轴回原点[M]
AND 2028.13  ; RK_05 U2_X #1入壳Y轴忙标志位
AND P_1s
LD H30.00  ; RK_05 U2_X #1入壳Y轴回原点记忆
ANDNOT 2028.13  ; RK_05 U2_X #1入壳Y轴忙标志位
ORLD
ANDLD
OUT 954.10  ; RK_05 U2_X #1入壳Y轴回原点[lamp]

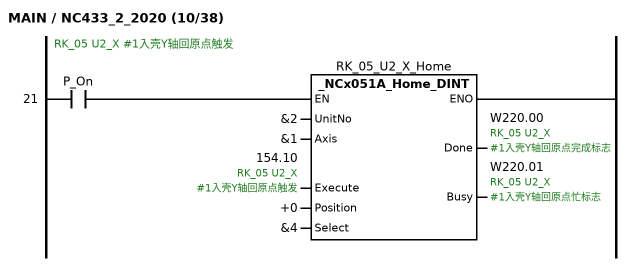
; rung 21: RK_05 U2_X #1入壳Y轴回原点触发
LD P_On
CALL RK_05_U2_X_Home : _NCx051A_Home_DINT (UnitNo := &2, Axis := &1, Execute := 154.10, Position := +0, Select := &4, Done => W220.00, Busy => W220.01)  ; RK_05 U2_X #1入壳Y轴回原点触发, RK_05 U2_X #1入壳Y轴回原点完成标志, RK_05 U2_X #1入壳Y轴回原点忙标志

